LIN {X 0,Y 358.362,Z 472.331,A -85,B 0,C 180,E1 -13392.156,E2 -13392.156} C_VEL
LIN {X 0,Y 357.855,Z 480.13,A -85,B 0,C 180,E1 -13393.015,E2 -13393.015} C_VEL
LIN {X 0,Y 356.562,Z 489.991,A -85,B 0,C 180,E1 -13394.276,E2 -13394.276} C_VEL
LIN {X 0,Y 355.505,Z 499.646,A -85,B 0,C 180,E1 -13395.781,E2 -13395.781} C_VEL
LIN {X 0,Y 355.018,Z 505.416,A -85,B 0,C 180,E1 -13396.841,E2 -13396.841} C_VEL
LIN {X 0,Y 354.311,Z 513.334,A -85,B 0,C 180,E1 -13398.559,E2 -13398.559} C_VEL
LIN {X 0,Y 353.919,Z 519.825,A -85,B 0,C 180,E1 -13400.283,E2 -13400.283} C_VEL
LIN {X 0,Y 353.818,Z 525.056,A -85,B 0,C 180,E1 -13402.008,E2 -13402.008} C_VEL
LIN {X 0,Y 353.937,Z 528.669,A -85,B 0,C 180,E1 -13403.503,E2 -13403.503} C_VEL
LIN {X 0,Y 354.156,Z 532.195,A -85,B 0,C 180,E1 -13405.447,E2 -13405.447} C_VEL
LIN {X 0,Y 354.254,Z 533.682,A -85,B 0,C 180,E1 -13406.588,E2 -13406.588} C_VEL
LIN {X 0,Y 354.319,Z 534.699,A -85,B 0,C 180,E1 -13407.727,E2 -13407.727} C_VEL
LIN {X 0,Y 354.65,Z 535.319,A -85,B 0,C 180,E1 -13408.865,E2 -13408.865} C_VEL
LIN {X 0,Y 354.78,Z 535.5,A -85,B 0,C 180,E1 -13410,E2 -13410} C_VEL
LIN {X 0,Y 354.651,Z 535.226,A -85,B 0,C 180,E1 -13411.135,E2 -13411.135} C_VEL
LIN {X 0,Y 354.359,Z 534.457,A -85,B 0,C 180,E1 -13412.273,E2 -13412.273} C_VEL
LIN {X 0,Y 354.31,Z 533.29,A -85,B 0,C 180,E1 -13413.411,E2 -13413.411} C_VEL
LIN {X 0,Y 354.165,Z 530.683,A -85,B 0,C 180,E1 -13415.123,E2 -13415.123} C_VEL
LIN {X 0,Y 353.996,Z 526.732,A -85,B 0,C 180,E1 -13416.941,E2 -13416.941} C_VEL
LIN {X 0,Y 353.922,Z 522.099,A -85,B 0,C 180,E1 -13418.565,E2 -13418.565} C_VEL
LIN {X 0,Y 354.064,Z 515.923,A -85,B 0,C 180,E1 -13420.291,E2 -13420.291} C_VEL
LIN {X 0,Y 354.504,Z 508.22,A -85,B 0,C 180,E1 -13422.014,E2 -13422.014} C_VEL
LIN {X 0,Y 355.133,Z 500.362,A -85,B 0,C 180,E1 -13423.446,E2 -13423.446} C_VEL
LIN {X 0,Y 355.912,Z 490.818,A -85,B 0,C 180,E1 -13424.874,E2 -13424.874} C_VEL
LIN {X 0,Y 356.895,Z 480.343,A -85,B 0,C 180,E1 -13426.149,E2 -13426.149} C_VEL
LIN {X 0,Y 357.392,Z 473.331,A -85,B 0,C 180,E1 -13426.861,E2 -13426.861} C_VEL
LIN {X 0,Y 356.949,Z 460.178,A -85,B 0,C 180,E1 -13427.991,E2 -13427.991} C_VEL
LIN {X 0,Y 356.126,Z 447.743,A -85,B 0,C 180,E1 -13428.815,E2 -13428.815} C_VEL
LIN {X 0,Y 354.927,Z 433.651,A -85,B 0,C 180,E1 -13429.509,E2 -13429.509} C_VEL
LIN {X 0,Y 354.262,Z 426.541,A -85,B 0,C 180,E1 -13429.822,E2 -13429.822} C_VEL
LIN {X 0,Y 354.936,Z 413.74,A -85,B 0,C 180,E1 -13433.879,E2 -13433.879} C_VEL
LIN {X 0,Y 355.803,Z 401.985,A -85,B 0,C 180,E1 -13437.703,E2 -13437.703} C_VEL
LIN {X 0,Y 356.859,Z 390.592,A -85,B 0,C 180,E1 -13441.458,E2 -13441.458} C_VEL
LIN {X 0,Y 358.142,Z 378.993,A -85,B 0,C 180,E1 -13445.372,E2 -13445.372} C_VEL
LIN {X 0,Y 358.881,Z 373.147,A -85,B 0,C 180,E1 -13447.377,E2 -13447.377} C_VEL
LIN {X 0,Y 357.713,Z 366.126,A -85,B 0,C 180,E1 -13449.983,E2 -13449.983} C_VEL
LIN {X 0,Y 355.825,Z 356.518,A -85,B 0,C 180,E1 -13453.731,E2 -13453.731} C_VEL
LIN {X 0,Y 354.834,Z 351.339,A -85,B 0,C 180,E1 -13455.939,E2 -13455.939} C_VEL
LIN {X 0,Y 354.76,Z 351.295,A -85,B 0,C 180,E1 -13459.175,E2 -13459.175} C_VEL
LIN {X 0,Y 354.795,Z 351.287,A -85,B 0,C 180,E1 -13462.403,E2 -13462.403} C_VEL
LIN {X 0,Y 354.806,Z 351.288,A -85,B 0,C 180,E1 -13464.94,E2 -13464.94} C_VEL
LIN {X 0,Y 354.787,Z 351.288,A -85,B 0,C 180,E1 -13468.405,E2 -13468.405} C_VEL
LIN {X 0,Y 354.843,Z 351.283,A -85,B 0,C 180,E1 -13471.618,E2 -13471.618} C_VEL
LIN {X 0,Y 354.891,Z 351.275,A -85,B 0,C 180,E1 -13474.172,E2 -13474.172} C_VEL
LIN {X 0,Y 354.808,Z 351.285,A -85,B 0,C 180,E1 -13477.892,E2 -13477.892} C_VEL
LIN {X 0,Y 354.882,Z 351.276,A -85,B 0,C 180,E1 -13481.908,E2 -13481.908} C_VEL
LIN {X 0,Y 354.934,Z 351.269,A -85,B 0,C 180,E1 -13485.981,E2 -13485.981} C_VEL
LIN {X 0,Y 354.947,Z 351.268,A -85,B 0,C 180,E1 -13489.735,E2 -13489.735} C_VEL
LIN {X 0,Y 355.102,Z 351.252,A -85,B 0,C 180,E1 -13493.18,E2 -13493.18} C_VEL
LIN {X 0,Y 355.234,Z 351.232,A -85,B 0,C 180,E1 -13497.732,E2 -13497.732} C_VEL
LIN {X 0,Y 355.388,Z 351.213,A -85,B 0,C 180,E1 -13500,E2 -13500} C_VEL
LIN {X 0,Y 355.233,Z 351.234,A -85,B 0,C 180,E1 -13502.268,E2 -13502.268} C_VEL
LIN {X 0,Y 355.118,Z 351.252,A -85,B 0,C 180,E1 -13506.82,E2 -13506.82} C_VEL
LIN {X 0,Y 354.969,Z 351.267,A -85,B 0,C 180,E1 -13510.264,E2 -13510.264} C_VEL
LIN {X 0,Y 354.934,Z 351.27,A -85,B 0,C 180,E1 -13514.019,E2 -13514.019} C_VEL
LIN {X 0,Y 354.915,Z 351.274,A -85,B 0,C 180,E1 -13518.109,E2 -13518.109} C_VEL
LIN {X 0,Y 354.828,Z 351.285,A -85,B 0,C 180,E1 -13522.107,E2 -13522.107} C_VEL
LIN {X 0,Y 354.892,Z 351.276,A -85,B 0,C 180,E1 -13525.828,E2 -13525.828} C_VEL
LIN {X 0,Y 354.848,Z 351.281,A -85,B 0,C 180,E1 -13529.679,E2 -13529.679} C_VEL
LIN {X 0,Y 354.8,Z 351.287,A -85,B 0,C 180,E1 -13533.703,E2 -13533.703} C_VEL
LIN {X 0,Y 354.794,Z 351.291,A -85,B 0,C 180,E1 -13536.46,E2 -13536.46} C_VEL
LIN {X 0,Y 354.819,Z 351.284,A -85,B 0,C 180,E1 -13539.424,E2 -13539.424} C_VEL
LIN {X 0,Y 354.8,Z 351.287,A -85,B 0,C 180,E1 -13542.871,E2 -13542.871} C_VEL
LIN {X 0,Y 354.772,Z 351.295,A -85,B 0,C 180,E1 -13546.106,E2 -13546.106} C_VEL
LIN {X 0,Y 354.788,Z 351.288,A -85,B 0,C 180,E1 -13549.18,E2 -13549.18} C_VEL
LIN {X 0,Y 354.806,Z 351.288,A -85,B 0,C 180,E1 -13552.403,E2 -13552.403} C_VEL
LIN {X 0,Y 354.811,Z 351.285,A -85,B 0,C 180,E1 -13554.942,E2 -13554.942} C_VEL
LIN {X 0,Y 354.814,Z 351.287,A -85,B 0,C 180,E1 -13558.4,E2 -13558.4} C_VEL
LIN {X 0,Y 354.853,Z 351.282,A -85,B 0,C 180,E1 -13561.62,E2 -13561.62} C_VEL
LIN {X 0,Y 354.899,Z 351.277,A -85,B 0,C 180,E1 -13564.173,E2 -13564.173} C_VEL
LIN {X 0,Y 354.835,Z 351.288,A -85,B 0,C 180,E1 -13567.895,E2 -13567.895} C_VEL
LIN {X 0,Y 354.924,Z 351.276,A -85,B 0,C 180,E1 -13571.892,E2 -13571.892} C_VEL
LIN {X 0,Y 354.944,Z 351.272,A -85,B 0,C 180,E1 -13575.981,E2 -13575.981} C_VEL
LIN {X 0,Y 354.98,Z 351.27,A -85,B 0,C 180,E1 -13579.736,E2 -13579.736} C_VEL
LIN {X 0,Y 355.116,Z 351.249,A -85,B 0,C 180,E1 -13582.037,E2 -13582.037} C_VEL
LIN {X 0,Y 355.096,Z 351.25,A -85,B 0,C 180,E1 -13584.321,E2 -13584.321} C_VEL
LIN {X 0,Y 355.248,Z 351.235,A -85,B 0,C 180,E1 -13587.732,E2 -13587.732} C_VEL
LIN {X 0,Y 355.4,Z 351.213,A -85,B 0,C 180,E1 -13590,E2 -13590} C_VEL
LIN {X 0,Y 355.249,Z 351.231,A -85,B 0,C 180,E1 -13592.268,E2 -13592.268} C_VEL
LIN {X 0,Y 355.127,Z 351.246,A -85,B 0,C 180,E1 -13596.819,E2 -13596.819} C_VEL
LIN {X 0,Y 354.98,Z 351.264,A -85,B 0,C 180,E1 -13600.264,E2 -13600.264} C_VEL
LIN {X 0,Y 354.944,Z 351.269,A -85,B 0,C 180,E1 -13604.019,E2 -13604.019} C_VEL
LIN {X 0,Y 354.923,Z 351.271,A -85,B 0,C 180,E1 -13608.108,E2 -13608.108} C_VEL
LIN {X 0,Y 354.835,Z 351.282,A -85,B 0,C 180,E1 -13612.105,E2 -13612.105} C_VEL
LIN {X 0,Y 354.899,Z 351.275,A -85,B 0,C 180,E1 -13615.827,E2 -13615.827} C_VEL
LIN {X 0,Y 354.817,Z 351.285,A -85,B 0,C 180,E1 -13619.681,E2 -13619.681} C_VEL
LIN {X 0,Y 354.804,Z 351.286,A -85,B 0,C 180,E1 -13623.701,E2 -13623.701} C_VEL
LIN {X 0,Y 354.8,Z 351.287,A -85,B 0,C 180,E1 -13626.458,E2 -13626.458} C_VEL
LIN {X 0,Y 354.821,Z 351.287,A -85,B 0,C 180,E1 -13629.423,E2 -13629.423} C_VEL
LIN {X 0,Y 354.863,Z 351.283,A -85,B 0,C 180,E1 -13632.88,E2 -13632.88} C_VEL
LIN {X 0,Y 354.916,Z 351.438,A -85,B 0,C 180,E1 -13633.417,E2 -13633.417} C_VEL
LIN {X 0,Y 355.205,Z 352.666,A -85,B 0,C 180,E1 -13633.637,E2 -13633.637} C_VEL
LIN {X 0,Y 358.7,Z 364.873,A -85,B 0,C 180,E1 -13634.725,E2 -13634.725} C_VEL
LIN {X 0,Y 360.105,Z 371.17,A -85,B 0,C 180,E1 -13635.364,E2 -13635.364} C_VEL
LIN {X 0,Y 359.332,Z 381.796,A -85,B 0,C 180,E1 -13636.463,E2 -13636.463} C_VEL
LIN {X 0,Y 358.503,Z 392.374,A -85,B 0,C 180,E1 -13637.823,E2 -13637.823} C_VEL
LIN {X 0,Y 357.866,Z 399.364,A -85,B 0,C 180,E1 -13638.893,E2 -13638.893} C_VEL
LIN {X 0,Y 356.907,Z 403.436,A -85,B 0,C 180,E1 -13639.571,E2 -13639.571} C_VEL
LIN {X 0,Y 353.622,Z 409.736,A -85,B 0,C 180,E1 -13640.678,E2 -13640.678} C_VEL
LIN {X 0,Y 350.29,Z 415.539,A -85,B 0,C 180,E1 -13641.869,E2 -13641.869} C_VEL
LIN {X 0,Y 349.276,Z 418.689,A -85,B 0,C 180,E1 -13642.67,E2 -13642.67} C_VEL
LIN {X 0,Y 348.734,Z 423.802,A -85,B 0,C 180,E1 -13644.237,E2 -13644.237} C_VEL
LIN {X 0,Y 348.313,Z 429.257,A -85,B 0,C 180,E1 -13646.391,E2 -13646.391} C_VEL
LIN {X 0,Y 348.034,Z 432.759,A -85,B 0,C 180,E1 -13648.33,E2 -13648.33} C_VEL
LIN {X 0,Y 347.912,Z 435.084,A -85,B 0,C 180,E1 -13650.296,E2 -13650.296} C_VEL
LIN {X 0,Y 347.965,Z 436.386,A -85,B 0,C 180,E1 -13652.706,E2 -13652.706} C_VEL
LIN {X 0,Y 348.247,Z 436.007,A -85,B 0,C 180,E1 -13654.925,E2 -13654.925} C_VEL
LIN {X 0,Y 348.528,Z 435.142,A -85,B 0,C 180,E1 -13656.216,E2 -13656.216} C_VEL
LIN {X 0,Y 348.981,Z 433.251,A -85,B 0,C 180,E1 -13657.873,E2 -13657.873} C_VEL
LIN {X 0,Y 349.767,Z 429.478,A -85,B 0,C 180,E1 -13660.026,E2 -13660.026} C_VEL
LIN {X 0,Y 350.61,Z 424.843,A -85,B 0,C 180,E1 -13661.899,E2 -13661.899} C_VEL
LIN {X 0,Y 351.666,Z 418.867,A -85,B 0,C 180,E1 -13663.752,E2 -13663.752} C_VEL
LIN {X 0,Y 352.692,Z 412.681,A -85,B 0,C 180,E1 -13665.282,E2 -13665.282} C_VEL
LIN {X 0,Y 353.995,Z 404.139,A -85,B 0,C 180,E1 -13666.984,E2 -13666.984} C_VEL
LIN {X 0,Y 355.367,Z 393.993,A -85,B 0,C 180,E1 -13668.594,E2 -13668.594} C_VEL
LIN {X 0,Y 356.593,Z 383.387,A -85,B 0,C 180,E1 -13669.928,E2 -13669.928} C_VEL
LIN {X 0,Y 357.097,Z 377.92,A -85,B 0,C 180,E1 -13670.512,E2 -13670.512} C_VEL
LIN {X 0,Y 353.861,Z 367.207,A -85,B 0,C 180,E1 -13671.865,E2 -13671.865} C_VEL
LIN {X 0,Y 350.27,Z 357.755,A -85,B 0,C 180,E1 -13672.941,E2 -13672.941} C_VEL
LIN {X 0,Y 348.165,Z 352.79,A -85,B 0,C 180,E1 -13673.517,E2 -13673.517} C_VEL
LIN {X 0,Y 348.064,Z 352.162,A -85,B 0,C 180,E1 -13673.769,E2 -13673.769} C_VEL
LIN {X 0,Y 348.196,Z 352.114,A -85,B 0,C 180,E1 -13677.686,E2 -13677.686} C_VEL
LIN {X 0,Y 348.337,Z 352.096,A -85,B 0,C 180,E1 -13680,E2 -13680} C_VEL
LIN {X 0,Y 348.196,Z 352.112,A -85,B 0,C 180,E1 -13682.314,E2 -13682.314} C_VEL
LIN {X 0,Y 348.068,Z 352.128,A -85,B 0,C 180,E1 -13686.958,E2 -13686.958} C_VEL
LIN {X 0,Y 347.887,Z 352.149,A -85,B 0,C 180,E1 -13690.476,E2 -13690.476} C_VEL
LIN {X 0,Y 347.891,Z 352.149,A -85,B 0,C 180,E1 -13694.15,E2 -13694.15} C_VEL
LIN {X 0,Y 347.821,Z 352.154,A -85,B 0,C 180,E1 -13698.26,E2 -13698.26} C_VEL
LIN {X 0,Y 347.76,Z 352.166,A -85,B 0,C 180,E1 -13701.627,E2 -13701.627} C_VEL
LIN {X 0,Y 347.805,Z 352.163,A -85,B 0,C 180,E1 -13705.109,E2 -13705.109} C_VEL
LIN {X 0,Y 347.802,Z 352.162,A -85,B 0,C 180,E1 -13707.695,E2 -13707.695} C_VEL
LIN {X 0,Y 347.743,Z 352.171,A -85,B 0,C 180,E1 -13710.349,E2 -13710.349} C_VEL
LIN {X 0,Y 347.743,Z 352.169,A -85,B 0,C 180,E1 -13714.045,E2 -13714.045} C_VEL
LIN {X 0,Y 347.751,Z 352.168,A -85,B 0,C 180,E1 -13717.322,E2 -13717.322} C_VEL
LIN {X 0,Y 347.734,Z 352.185,A -85,B 0,C 180,E1 -13721.601,E2 -13721.601} C_VEL
LIN {X 0,Y 348.038,Z 353.526,A -85,B 0,C 180,E1 -13722.569,E2 -13722.569} C_VEL
LIN {X 0,Y 349.523,Z 360.428,A -85,B 0,C 180,E1 -13726.375,E2 -13726.375} C_VEL
LIN {X 0,Y 351.027,Z 368.334,A -85,B 0,C 180,E1 -13730.159,E2 -13730.159} C_VEL
LIN {X 0,Y 351.776,Z 373.684,A -85,B 0,C 180,E1 -13732.46,E2 -13732.46} C_VEL
LIN {X 0,Y 350.204,Z 384.504,A -85,B 0,C 180,E1 -13736.505,E2 -13736.505} C_VEL
LIN {X 0,Y 349.147,Z 394.206,A -85,B 0,C 180,E1 -13739.946,E2 -13739.946} C_VEL
LIN {X 0,Y 348.219,Z 405.075,A -85,B 0,C 180,E1 -13743.64,E2 -13743.64} C_VEL
LIN {X 0,Y 347.447,Z 417.359,A -85,B 0,C 180,E1 -13747.625,E2 -13747.625} C_VEL
LIN {X 0,Y 347.592,Z 419.174,A -85,B 0,C 180,E1 -13747.812,E2 -13747.812} C_VEL
LIN {X 0,Y 350.112,Z 432.508,A -85,B 0,C 180,E1 -13748.583,E2 -13748.583} C_VEL
LIN {X 0,Y 351.458,Z 445.441,A -85,B 0,C 180,E1 -13749.441,E2 -13749.441} C_VEL
LIN {X 0,Y 351.882,Z 457.391,A -85,B 0,C 180,E1 -13750.379,E2 -13750.379} C_VEL
LIN {X 0,Y 351.551,Z 469.302,A -85,B 0,C 180,E1 -13751.497,E2 -13751.497} C_VEL
LIN {X 0,Y 351.215,Z 478.527,A -85,B 0,C 180,E1 -13752.533,E2 -13752.533} C_VEL
LIN {X 0,Y 349.667,Z 489.454,A -85,B 0,C 180,E1 -13753.957,E2 -13753.957} C_VEL
LIN {X 0,Y 348.568,Z 498.626,A -85,B 0,C 180,E1 -13755.421,E2 -13755.421} C_VEL
LIN {X 0,Y 348.085,Z 504.722,A -85,B 0,C 180,E1 -13756.574,E2 -13756.574} C_VEL
LIN {X 0,Y 347.306,Z 512.567,A -85,B 0,C 180,E1 -13758.325,E2 -13758.325} C_VEL
LIN {X 0,Y 346.847,Z 518.982,A -85,B 0,C 180,E1 -13760.083,E2 -13760.083} C_VEL
LIN {X 0,Y 346.74,Z 524.165,A -85,B 0,C 180,E1 -13761.843,E2 -13761.843} C_VEL
LIN {X 0,Y 346.825,Z 527.351,A -85,B 0,C 180,E1 -13763.183,E2 -13763.183} C_VEL
LIN {X 0,Y 347.091,Z 531.243,A -85,B 0,C 180,E1 -13765.354,E2 -13765.354} C_VEL
LIN {X 0,Y 347.203,Z 532.71,A -85,B 0,C 180,E1 -13766.519,E2 -13766.519} C_VEL
LIN {X 0,Y 347.617,Z 534.301,A -85,B 0,C 180,E1 -13768.842,E2 -13768.842} C_VEL
LIN {X 0,Y 347.772,Z 534.47,A -85,B 0,C 180,E1 -13770,E2 -13770} C_VEL
LIN {X 0,Y 347.621,Z 534.165,A -85,B 0,C 180,E1 -13771.158,E2 -13771.158} C_VEL
LIN {X 0,Y 347.27,Z 532.179,A -85,B 0,C 180,E1 -13773.481,E2 -13773.481} C_VEL
LIN {X 0,Y 347.108,Z 529.527,A -85,B 0,C 180,E1 -13775.228,E2 -13775.228} C_VEL
LIN {X 0,Y 346.945,Z 525.775,A -85,B 0,C 180,E1 -13776.981,E2 -13776.981} C_VEL
LIN {X 0,Y 346.874,Z 520.839,A -85,B 0,C 180,E1 -13778.74,E2 -13778.74} C_VEL
LIN {X 0,Y 347.015,Z 514.6,A -85,B 0,C 180,E1 -13780.502,E2 -13780.502} C_VEL
LIN {X 0,Y 347.491,Z 506.787,A -85,B 0,C 180,E1 -13782.261,E2 -13782.261} C_VEL
LIN {X 0,Y 348.101,Z 498.832,A -85,B 0,C 180,E1 -13783.723,E2 -13783.723} C_VEL
LIN {X 0,Y 348.98,Z 489.198,A -85,B 0,C 180,E1 -13785.177,E2 -13785.177} C_VEL
LIN {X 0,Y 350.007,Z 478.575,A -85,B 0,C 180,E1 -13786.476,E2 -13786.476} C_VEL
LIN {X 0,Y 350.321,Z 472.921,A -85,B 0,C 180,E1 -13787.061,E2 -13787.061} C_VEL
LIN {X 0,Y 349.964,Z 460.881,A -85,B 0,C 180,E1 -13788.135,E2 -13788.135} C_VEL
LIN {X 0,Y 349.245,Z 449.494,A -85,B 0,C 180,E1 -13788.95,E2 -13788.95} C_VEL
LIN {X 0,Y 348.207,Z 435.937,A -85,B 0,C 180,E1 -13789.682,E2 -13789.682} C_VEL
LIN {X 0,Y 347.223,Z 425.817,A -85,B 0,C 180,E1 -13790.126,E2 -13790.126} C_VEL
LIN {X 0,Y 347.596,Z 418.073,A -85,B 0,C 180,E1 -13792.591,E2 -13792.591} C_VEL
LIN {X 0,Y 348.391,Z 406.693,A -85,B 0,C 180,E1 -13796.346,E2 -13796.346} C_VEL
LIN {X 0,Y 349.398,Z 395.257,A -85,B 0,C 180,E1 -13800.189,E2 -13800.189} C_VEL
LIN {X 0,Y 350.427,Z 385.651,A -85,B 0,C 180,E1 -13803.471,E2 -13803.471} C_VEL
LIN {X 0,Y 351.762,Z 375.625,A -85,B 0,C 180,E1 -13806.948,E2 -13806.948} C_VEL
LIN {X 0,Y 351.777,Z 372.982,A -85,B 0,C 180,E1 -13807.904,E2 -13807.904} C_VEL
LIN {X 0,Y 350.001,Z 363.655,A -85,B 0,C 180,E1 -13811.5,E2 -13811.5} C_VEL
LIN {X 0,Y 348.319,Z 354.848,A -85,B 0,C 180,E1 -13815.074,E2 -13815.074} C_VEL
LIN {X 0,Y 347.758,Z 352.252,A -85,B 0,C 180,E1 -13816.197,E2 -13816.197} C_VEL
LIN {X 0,Y 347.692,Z 352.174,A -85,B 0,C 180,E1 -13819.697,E2 -13819.697} C_VEL
LIN {X 0,Y 347.751,Z 352.165,A -85,B 0,C 180,E1 -13822.678,E2 -13822.678} C_VEL
LIN {X 0,Y 347.743,Z 352.166,A -85,B 0,C 180,E1 -13825.955,E2 -13825.955} C_VEL
LIN {X 0,Y 347.758,Z 352.165,A -85,B 0,C 180,E1 -13829.653,E2 -13829.653} C_VEL
LIN {X 0,Y 347.844,Z 352.155,A -85,B 0,C 180,E1 -13832.744,E2 -13832.744} C_VEL
LIN {X 0,Y 347.778,Z 352.161,A -85,B 0,C 180,E1 -13836.161,E2 -13836.161} C_VEL
LIN {X 0,Y 347.792,Z 352.159,A -85,B 0,C 180,E1 -13839.908,E2 -13839.908} C_VEL
LIN {X 0,Y 347.824,Z 352.157,A -85,B 0,C 180,E1 -13843.568,E2 -13843.568} C_VEL
LIN {X 0,Y 347.881,Z 352.152,A -85,B 0,C 180,E1 -13847.16,E2 -13847.16} C_VEL
LIN {X 0,Y 347.927,Z 352.146,A -85,B 0,C 180,E1 -13850.7,E2 -13850.7} C_VEL
LIN {X 0,Y 348.068,Z 352.129,A -85,B 0,C 180,E1 -13853.042,E2 -13853.042} C_VEL
LIN {X 0,Y 348.196,Z 352.109,A -85,B 0,C 180,E1 -13857.686,E2 -13857.686} C_VEL
LIN {X 0,Y 348.337,Z 352.091,A -85,B 0,C 180,E1 -13860,E2 -13860} C_VEL
LIN {X 0,Y 348.196,Z 352.111,A -85,B 0,C 180,E1 -13862.314,E2 -13862.314} C_VEL
LIN {X 0,Y 348.084,Z 352.126,A -85,B 0,C 180,E1 -13866.958,E2 -13866.958} C_VEL
LIN {X 0,Y 347.92,Z 352.147,A -85,B 0,C 180,E1 -13870.475,E2 -13870.475} C_VEL
LIN {X 0,Y 347.891,Z 352.149,A -85,B 0,C 180,E1 -13874.15,E2 -13874.15} C_VEL
LIN {X 0,Y 347.884,Z 352.151,A -85,B 0,C 180,E1 -13878.291,E2 -13878.291} C_VEL
LIN {X 0,Y 347.782,Z 352.16,A -85,B 0,C 180,E1 -13881.636,E2 -13881.636} C_VEL
LIN {X 0,Y 347.805,Z 352.158,A -85,B 0,C 180,E1 -13885.109,E2 -13885.109} C_VEL
LIN {X 0,Y 347.806,Z 352.158,A -85,B 0,C 180,E1 -13887.694,E2 -13887.694} C_VEL
LIN {X 0,Y 347.758,Z 352.169,A -85,B 0,C 180,E1 -13890.347,E2 -13890.347} C_VEL
LIN {X 0,Y 347.739,Z 352.17,A -85,B 0,C 180,E1 -13894.465,E2 -13894.465} C_VEL
LIN {X 0,Y 347.77,Z 352.165,A -85,B 0,C 180,E1 -13897.99,E2 -13897.99} C_VEL
LIN {X 0,Y 347.762,Z 352.165,A -85,B 0,C 180,E1 -13901.829,E2 -13901.829} C_VEL
LIN {X 0,Y 347.73,Z 352.167,A -85,B 0,C 180,E1 -13905.023,E2 -13905.023} C_VEL
LIN {X 0,Y 347.75,Z 352.168,A -85,B 0,C 180,E1 -13908.397,E2 -13908.397} C_VEL
LIN {X 0,Y 347.772,Z 352.167,A -85,B 0,C 180,E1 -13912.012,E2 -13912.012} C_VEL
LIN {X 0,Y 347.743,Z 352.167,A -85,B 0,C 180,E1 -13915.537,E2 -13915.537} C_VEL
LIN {X 0,Y 347.763,Z 352.166,A -85,B 0,C 180,E1 -13918.303,E2 -13918.303} C_VEL
LIN {X 0,Y 347.805,Z 352.157,A -85,B 0,C 180,E1 -13920.991,E2 -13920.991} C_VEL
LIN {X 0,Y 347.832,Z 352.157,A -85,B 0,C 180,E1 -13923.609,E2 -13923.609} C_VEL
LIN {X 0,Y 347.789,Z 352.163,A -85,B 0,C 180,E1 -13926.163,E2 -13926.163} C_VEL
LIN {X 0,Y 347.818,Z 352.161,A -85,B 0,C 180,E1 -13929.91,E2 -13929.91} C_VEL
LIN {X 0,Y 347.868,Z 352.151,A -85,B 0,C 180,E1 -13932.36,E2 -13932.36} C_VEL
LIN {X 0,Y 347.899,Z 352.15,A -85,B 0,C 180,E1 -13935.971,E2 -13935.971} C_VEL
LIN {X 0,Y 347.931,Z 352.146,A -85,B 0,C 180,E1 -13939.526,E2 -13939.526} C_VEL
LIN {X 0,Y 348.077,Z 352.128,A -85,B 0,C 180,E1 -13941.875,E2 -13941.875} C_VEL
LIN {X 0,Y 348.071,Z 352.125,A -85,B 0,C 180,E1 -13944.206,E2 -13944.206} C_VEL
LIN {X 0,Y 348.211,Z 352.112,A -85,B 0,C 180,E1 -13947.687,E2 -13947.687} C_VEL
LIN {X 0,Y 348.37,Z 352.089,A -85,B 0,C 180,E1 -13950,E2 -13950} C_VEL
LIN {X 0,Y 348.211,Z 352.107,A -85,B 0,C 180,E1 -13952.313,E2 -13952.313} C_VEL
LIN {X 0,Y 348.093,Z 352.123,A -85,B 0,C 180,E1 -13956.958,E2 -13956.958} C_VEL
LIN {X 0,Y 347.931,Z 352.142,A -85,B 0,C 180,E1 -13960.474,E2 -13960.474} C_VEL
LIN {X 0,Y 347.9,Z 352.146,A -85,B 0,C 180,E1 -13964.149,E2 -13964.149} C_VEL
LIN {X 0,Y 347.891,Z 352.147,A -85,B 0,C 180,E1 -13968.29,E2 -13968.29} C_VEL
LIN {X 0,Y 347.789,Z 352.162,A -85,B 0,C 180,E1 -13971.635,E2 -13971.635} C_VEL
LIN {X 0,Y 347.813,Z 352.162,A -85,B 0,C 180,E1 -13975.108,E2 -13975.108} C_VEL
LIN {X 0,Y 347.807,Z 352.159,A -85,B 0,C 180,E1 -13977.693,E2 -13977.693} C_VEL
LIN {X 0,Y 347.748,Z 352.165,A -85,B 0,C 180,E1 -13980.347,E2 -13980.347} C_VEL
LIN {X 0,Y 347.746,Z 352.165,A -85,B 0,C 180,E1 -13984.043,E2 -13984.043} C_VEL
LIN {X 0,Y 347.765,Z 352.166,A -85,B 0,C 180,E1 -13987.319,E2 -13987.319} C_VEL
LIN {X 0,Y 347.791,Z 352.164,A -85,B 0,C 180,E1 -13990.288,E2 -13990.288} C_VEL
LIN {X 0,Y 347.848,Z 352.299,A -85,B 0,C 180,E1 -13993.111,E2 -13993.111} C_VEL
LIN {X 0,Y 348.15,Z 353.58,A -85,B 0,C 180,E1 -13993.34,E2 -13993.34} C_VEL
LIN {X 0,Y 351.892,Z 366.568,A -85,B 0,C 180,E1 -13994.531,E2 -13994.531} C_VEL
LIN {X 0,Y 353.126,Z 371.448,A -85,B 0,C 180,E1 -13995.043,E2 -13995.043} C_VEL
LIN {X 0,Y 352.491,Z 382.216,A -85,B 0,C 180,E1 -13996.173,E2 -13996.173} C_VEL
LIN {X 0,Y 351.656,Z 392.654,A -85,B 0,C 180,E1 -13997.519,E2 -13997.519} C_VEL
LIN {X 0,Y 350.66,Z 403.079,A -85,B 0,C 180,E1 -13999.195,E2 -13999.195} C_VEL
LIN {X 0,Y 349.942,Z 410.961,A -85,B 0,C 180,E1 -14000.756,E2 -14000.756} C_VEL
LIN {X 0,Y 349.276,Z 418.689,A -85,B 0,C 180,E1 -14002.67,E2 -14002.67} C_VEL
LIN {X 0,Y 348.284,Z 421.652,A -85,B 0,C 180,E1 -14003.496,E2 -14003.496} C_VEL
LIN {X 0,Y 345.055,Z 426.138,A -85,B 0,C 180,E1 -14004.857,E2 -14004.857} C_VEL
LIN {X 0,Y 341.939,Z 429.996,A -85,B 0,C 180,E1 -14006.291,E2 -14006.291} C_VEL
LIN {X 0,Y 341.141,Z 431.89,A -85,B 0,C 180,E1 -14007.22,E2 -14007.22} C_VEL
LIN {X 0,Y 340.934,Z 434.654,A -85,B 0,C 180,E1 -14008.979,E2 -14008.979} C_VEL
LIN {X 0,Y 340.892,Z 436.108,A -85,B 0,C 180,E1 -14010.344,E2 -14010.344} C_VEL
LIN {X 0,Y 340.932,Z 437.318,A -85,B 0,C 180,E1 -14012.422,E2 -14012.422} C_VEL
LIN {X 0,Y 341.25,Z 437.113,A -85,B 0,C 180,E1 -14014.979,E2 -14014.979} C_VEL
LIN {X 0,Y 341.72,Z 435.618,A -85,B 0,C 180,E1 -14016.998,E2 -14016.998} C_VEL
LIN {X 0,Y 342.378,Z 433.031,A -85,B 0,C 180,E1 -14018.947,E2 -14018.947} C_VEL
LIN {X 0,Y 343.134,Z 429.312,A -85,B 0,C 180,E1 -14020.87,E2 -14020.87} C_VEL
LIN {X 0,Y 344.15,Z 424.285,A -85,B 0,C 180,E1 -14022.776,E2 -14022.776} C_VEL
LIN {X 0,Y 345.316,Z 417.835,A -85,B 0,C 180,E1 -14024.658,E2 -14024.658} C_VEL
LIN {X 0,Y 346.607,Z 410.454,A -85,B 0,C 180,E1 -14026.366,E2 -14026.366} C_VEL
LIN {X 0,Y 347.695,Z 403.174,A -85,B 0,C 180,E1 -14027.746,E2 -14027.746} C_VEL
LIN {X 0,Y 349.151,Z 393.29,A -85,B 0,C 180,E1 -14029.269,E2 -14029.269} C_VEL
LIN {X 0,Y 350.355,Z 383.05,A -85,B 0,C 180,E1 -14030.547,E2 -14030.547} C_VEL
LIN {X 0,Y 350.561,Z 379.755,A -85,B 0,C 180,E1 -14030.916,E2 -14030.916} C_VEL
LIN {X 0,Y 347.544,Z 369.665,A -85,B 0,C 180,E1 -14032.243,E2 -14032.243} C_VEL
LIN {X 0,Y 343.446,Z 358.895,A -85,B 0,C 180,E1 -14033.538,E2 -14033.538} C_VEL
LIN {X 0,Y 341.156,Z 353.736,A -85,B 0,C 180,E1 -14034.162,E2 -14034.162} C_VEL
LIN {X 0,Y 340.96,Z 353.046,A -85,B 0,C 180,E1 -14034.455,E2 -14034.455} C_VEL
LIN {X 0,Y 341.158,Z 352.99,A -85,B 0,C 180,E1 -14037.639,E2 -14037.639} C_VEL
LIN {X 0,Y 341.287,Z 352.975,A -85,B 0,C 180,E1 -14040,E2 -14040} C_VEL
LIN {X 0,Y 341.158,Z 352.989,A -85,B 0,C 180,E1 -14042.361,E2 -14042.361} C_VEL
LIN {X 0,Y 341.036,Z 353.005,A -85,B 0,C 180,E1 -14047.103,E2 -14047.103} C_VEL
LIN {X 0,Y 340.839,Z 353.028,A -85,B 0,C 180,E1 -14050.695,E2 -14050.695} C_VEL
LIN {X 0,Y 340.856,Z 353.026,A -85,B 0,C 180,E1 -14054.325,E2 -14054.325} C_VEL
LIN {X 0,Y 340.779,Z 353.032,A -85,B 0,C 180,E1 -14058.441,E2 -14058.441} C_VEL
LIN {X 0,Y 340.711,Z 353.045,A -85,B 0,C 180,E1 -14061.842,E2 -14061.842} C_VEL
LIN {X 0,Y 340.765,Z 353.036,A -85,B 0,C 180,E1 -14065.665,E2 -14065.665} C_VEL
LIN {X 0,Y 340.722,Z 353.042,A -85,B 0,C 180,E1 -14068.321,E2 -14068.321} C_VEL
LIN {X 0,Y 340.691,Z 353.045,A -85,B 0,C 180,E1 -14071.045,E2 -14071.045} C_VEL
LIN {X 0,Y 340.712,Z 353.043,A -85,B 0,C 180,E1 -14075.28,E2 -14075.28} C_VEL
LIN {X 0,Y 340.688,Z 353.048,A -85,B 0,C 180,E1 -14078.383,E2 -14078.383} C_VEL
LIN {X 0,Y 340.688,Z 353.171,A -85,B 0,C 180,E1 -14081.015,E2 -14081.015} C_VEL
LIN {X 0,Y 341.886,Z 358.639,A -85,B 0,C 180,E1 -14084.341,E2 -14084.341} C_VEL
LIN {X 0,Y 343.106,Z 364.605,A -85,B 0,C 180,E1 -14087.511,E2 -14087.511} C_VEL
LIN {X 0,Y 344.414,Z 371.625,A -85,B 0,C 180,E1 -14090.843,E2 -14090.843} C_VEL
LIN {X 0,Y 344.845,Z 374.984,A -85,B 0,C 180,E1 -14092.31,E2 -14092.31} C_VEL
LIN {X 0,Y 343.225,Z 385.747,A -85,B 0,C 180,E1 -14096.437,E2 -14096.437} C_VEL
LIN {X 0,Y 341.96,Z 396.829,A -85,B 0,C 180,E1 -14100.446,E2 -14100.446} C_VEL
LIN {X 0,Y 340.994,Z 408.119,A -85,B 0,C 180,E1 -14104.354,E2 -14104.354} C_VEL
LIN {X 0,Y 340.457,Z 416.172,A -85,B 0,C 180,E1 -14107.005,E2 -14107.005} C_VEL
LIN {X 0,Y 340.648,Z 418.024,A -85,B 0,C 180,E1 -14107.171,E2 -14107.171} C_VEL
LIN {X 0,Y 343.135,Z 430.572,A -85,B 0,C 180,E1 -14107.933,E2 -14107.933} C_VEL
LIN {X 0,Y 344.667,Z 443.838,A -85,B 0,C 180,E1 -14108.86,E2 -14108.86} C_VEL
LIN {X 0,Y 345.119,Z 456.528,A -85,B 0,C 180,E1 -14109.884,E2 -14109.884} C_VEL
LIN {X 0,Y 344.816,Z 467.8,A -85,B 0,C 180,E1 -14110.968,E2 -14110.968} C_VEL
LIN {X 0,Y 344.26,Z 479.412,A -85,B 0,C 180,E1 -14112.322,E2 -14112.322} C_VEL
LIN {X 0,Y 342.839,Z 488.987,A -85,B 0,C 180,E1 -14113.629,E2 -14113.629} C_VEL
LIN {X 0,Y 341.569,Z 498.748,A -85,B 0,C 180,E1 -14115.253,E2 -14115.253} C_VEL
LIN {X 0,Y 340.929,Z 505.454,A -85,B 0,C 180,E1 -14116.591,E2 -14116.591} C_VEL
LIN {X 0,Y 340.177,Z 512.982,A -85,B 0,C 180,E1 -14118.38,E2 -14118.38} C_VEL
LIN {X 0,Y 339.713,Z 519.993,A -85,B 0,C 180,E1 -14120.474,E2 -14120.474} C_VEL
LIN {X 0,Y 339.675,Z 524.738,A -85,B 0,C 180,E1 -14122.271,E2 -14122.271} C_VEL
LIN {X 0,Y 339.829,Z 528.4,A -85,B 0,C 180,E1 -14124.065,E2 -14124.065} C_VEL
LIN {X 0,Y 340.027,Z 530.291,A -85,B 0,C 180,E1 -14125.258,E2 -14125.258} C_VEL
LIN {X 0,Y 340.153,Z 531.729,A -85,B 0,C 180,E1 -14126.446,E2 -14126.446} C_VEL
LIN {X 0,Y 340.583,Z 533.288,A -85,B 0,C 180,E1 -14128.818,E2 -14128.818} C_VEL
LIN {X 0,Y 340.762,Z 533.443,A -85,B 0,C 180,E1 -14130,E2 -14130} C_VEL
LIN {X 0,Y 340.59,Z 533.093,A -85,B 0,C 180,E1 -14131.182,E2 -14131.182} C_VEL
LIN {X 0,Y 340.229,Z 531.066,A -85,B 0,C 180,E1 -14133.553,E2 -14133.553} C_VEL
LIN {X 0,Y 340.052,Z 528.364,A -85,B 0,C 180,E1 -14135.336,E2 -14135.336} C_VEL
LIN {X 0,Y 339.877,Z 524.558,A -85,B 0,C 180,E1 -14137.127,E2 -14137.127} C_VEL
LIN {X 0,Y 339.806,Z 519.565,A -85,B 0,C 180,E1 -14138.923,E2 -14138.923} C_VEL
LIN {X 0,Y 339.996,Z 513.256,A -85,B 0,C 180,E1 -14140.721,E2 -14140.721} C_VEL
LIN {X 0,Y 340.489,Z 505.34,A -85,B 0,C 180,E1 -14142.517,E2 -14142.517} C_VEL
LIN {X 0,Y 341.099,Z 497.292,A -85,B 0,C 180,E1 -14144.01,E2 -14144.01} C_VEL
LIN {X 0,Y 342.102,Z 487.58,A -85,B 0,C 180,E1 -14145.489,E2 -14145.489} C_VEL
LIN {X 0,Y 343.213,Z 476.771,A -85,B 0,C 180,E1 -14146.812,E2 -14146.812} C_VEL
LIN {X 0,Y 343.116,Z 466.062,A -85,B 0,C 180,E1 -14147.893,E2 -14147.893} C_VEL
LIN {X 0,Y 342.501,Z 452.954,A -85,B 0,C 180,E1 -14148.959,E2 -14148.959} C_VEL
LIN {X 0,Y 341.51,Z 439.372,A -85,B 0,C 180,E1 -14149.791,E2 -14149.791} C_VEL
LIN {X 0,Y 340.184,Z 425.2,A -85,B 0,C 180,E1 -14150.442,E2 -14150.442} C_VEL
LIN {X 0,Y 340.176,Z 424.448,A -85,B 0,C 180,E1 -14150.561,E2 -14150.561} C_VEL
LIN {X 0,Y 340.849,Z 413.1,A -85,B 0,C 180,E1 -14154.354,E2 -14154.354} C_VEL
LIN {X 0,Y 341.777,Z 401.75,A -85,B 0,C 180,E1 -14158.225,E2 -14158.225} C_VEL
LIN {X 0,Y 342.945,Z 390.289,A -85,B 0,C 180,E1 -14162.195,E2 -14162.195} C_VEL
LIN {X 0,Y 344.636,Z 377.243,A -85,B 0,C 180,E1 -14166.815,E2 -14166.815} C_VEL
LIN {X 0,Y 344.851,Z 374.832,A -85,B 0,C 180,E1 -14167.689,E2 -14167.689} C_VEL
LIN {X 0,Y 343.352,Z 366.552,A -85,B 0,C 180,E1 -14170.918,E2 -14170.918} C_VEL
LIN {X 0,Y 341.719,Z 358.123,A -85,B 0,C 180,E1 -14174.367,E2 -14174.367} C_VEL
LIN {X 0,Y 340.724,Z 353.12,A -85,B 0,C 180,E1 -14176.557,E2 -14176.557} C_VEL
LIN {X 0,Y 340.65,Z 353.049,A -85,B 0,C 180,E1 -14180.24,E2 -14180.24} C_VEL
LIN {X 0,Y 340.703,Z 353.046,A -85,B 0,C 180,E1 -14183.559,E2 -14183.559} C_VEL
LIN {X 0,Y 340.687,Z 353.044,A -85,B 0,C 180,E1 -14186.153,E2 -14186.153} C_VEL
LIN {X 0,Y 340.768,Z 353.034,A -85,B 0,C 180,E1 -14190.332,E2 -14190.332} C_VEL
LIN {X 0,Y 340.797,Z 353.035,A -85,B 0,C 180,E1 -14193.019,E2 -14193.019} C_VEL
LIN {X 0,Y 340.747,Z 353.038,A -85,B 0,C 180,E1 -14195.638,E2 -14195.638} C_VEL
LIN {X 0,Y 340.722,Z 353.042,A -85,B 0,C 180,E1 -14199.472,E2 -14199.472} C_VEL
LIN {X 0,Y 340.784,Z 353.032,A -85,B 0,C 180,E1 -14201.98,E2 -14201.98} C_VEL
LIN {X 0,Y 340.862,Z 353.023,A -85,B 0,C 180,E1 -14205.705,E2 -14205.705} C_VEL
LIN {X 0,Y 340.839,Z 353.028,A -85,B 0,C 180,E1 -14209.305,E2 -14209.305} C_VEL
LIN {X 0,Y 341.036,Z 353.007,A -85,B 0,C 180,E1 -14212.897,E2 -14212.897} C_VEL
LIN {X 0,Y 341.158,Z 352.986,A -85,B 0,C 180,E1 -14217.639,E2 -14217.639} C_VEL
LIN {X 0,Y 341.287,Z 352.97,A -85,B 0,C 180,E1 -14220,E2 -14220} C_VEL
LIN {X 0,Y 341.157,Z 352.988,A -85,B 0,C 180,E1 -14222.361,E2 -14222.361} C_VEL
LIN {X 0,Y 341.052,Z 353.001,A -85,B 0,C 180,E1 -14227.102,E2 -14227.102} C_VEL
LIN {X 0,Y 340.862,Z 353.028,A -85,B 0,C 180,E1 -14230.694,E2 -14230.694} C_VEL
LIN {X 0,Y 340.856,Z 353.026,A -85,B 0,C 180,E1 -14234.325,E2 -14234.325} C_VEL
LIN {X 0,Y 340.831,Z 353.032,A -85,B 0,C 180,E1 -14238.467,E2 -14238.467} C_VEL
LIN {X 0,Y 340.747,Z 353.038,A -85,B 0,C 180,E1 -14241.857,E2 -14241.857} C_VEL
LIN {X 0,Y 340.766,Z 353.035,A -85,B 0,C 180,E1 -14245.665,E2 -14245.665} C_VEL
LIN {X 0,Y 340.736,Z 353.043,A -85,B 0,C 180,E1 -14248.32,E2 -14248.32} C_VEL
LIN {X 0,Y 340.698,Z 353.043,A -85,B 0,C 180,E1 -14251.045,E2 -14251.045} C_VEL
LIN {X 0,Y 340.713,Z 353.041,A -85,B 0,C 180,E1 -14255.28,E2 -14255.28} C_VEL
LIN {X 0,Y 340.708,Z 353.046,A -85,B 0,C 180,E1 -14258.387,E2 -14258.387} C_VEL
LIN {X 0,Y 340.725,Z 353.044,A -85,B 0,C 180,E1 -14262.052,E2 -14262.052} C_VEL
LIN {X 0,Y 340.658,Z 353.053,A -85,B 0,C 180,E1 -14266.226,E2 -14266.226} C_VEL
LIN {X 0,Y 340.688,Z 353.047,A -85,B 0,C 180,E1 -14269.753,E2 -14269.753} C_VEL
LIN {X 0,Y 340.703,Z 353.042,A -85,B 0,C 180,E1 -14273.259,E2 -14273.259} C_VEL
LIN {X 0,Y 340.694,Z 353.048,A -85,B 0,C 180,E1 -14276.154,E2 -14276.154} C_VEL
LIN {X 0,Y 340.775,Z 353.036,A -85,B 0,C 180,E1 -14280.333,E2 -14280.333} C_VEL
LIN {X 0,Y 340.805,Z 353.03,A -85,B 0,C 180,E1 -14283.021,E2 -14283.021} C_VEL
LIN {X 0,Y 340.729,Z 353.039,A -85,B 0,C 180,E1 -14286.928,E2 -14286.928} C_VEL
LIN {X 0,Y 340.796,Z 353.031,A -85,B 0,C 180,E1 -14290.734,E2 -14290.734} C_VEL
LIN {X 0,Y 340.789,Z 353.033,A -85,B 0,C 180,E1 -14293.219,E2 -14293.219} C_VEL
LIN {X 0,Y 340.846,Z 353.025,A -85,B 0,C 180,E1 -14296.891,E2 -14296.891} C_VEL
LIN {X 0,Y 340.93,Z 353.014,A -85,B 0,C 180,E1 -14300.508,E2 -14300.508} C_VEL
LIN {X 0,Y 341.078,Z 352.996,A -85,B 0,C 180,E1 -14302.898,E2 -14302.898} C_VEL
LIN {X 0,Y 341.172,Z 352.989,A -85,B 0,C 180,E1 -14307.639,E2 -14307.639} C_VEL
LIN {X 0,Y 341.319,Z 352.967,A -85,B 0,C 180,E1 -14310,E2 -14310} C_VEL
LIN {X 0,Y 341.173,Z 352.984,A -85,B 0,C 180,E1 -14312.361,E2 -14312.361} C_VEL
LIN {X 0,Y 341.061,Z 353,A -85,B 0,C 180,E1 -14317.102,E2 -14317.102} C_VEL
LIN {X 0,Y 340.873,Z 353.022,A -85,B 0,C 180,E1 -14320.693,E2 -14320.693} C_VEL
LIN {X 0,Y 340.864,Z 353.022,A -85,B 0,C 180,E1 -14324.324,E2 -14324.324} C_VEL
LIN {X 0,Y 340.838,Z 353.026,A -85,B 0,C 180,E1 -14328.466,E2 -14328.466} C_VEL
LIN {X 0,Y 340.754,Z 353.037,A -85,B 0,C 180,E1 -14331.856,E2 -14331.856} C_VEL
LIN {X 0,Y 340.772,Z 353.035,A -85,B 0,C 180,E1 -14335.664,E2 -14335.664} C_VEL
LIN {X 0,Y 340.728,Z 353.039,A -85,B 0,C 180,E1 -14338.32,E2 -14338.32} C_VEL
LIN {X 0,Y 340.696,Z 353.049,A -85,B 0,C 180,E1 -14341.044,E2 -14341.044} C_VEL
LIN {X 0,Y 340.717,Z 353.044,A -85,B 0,C 180,E1 -14345.278,E2 -14345.278} C_VEL
LIN {X 0,Y 340.717,Z 353.041,A -85,B 0,C 180,E1 -14348.387,E2 -14348.387} C_VEL
LIN {X 0,Y 340.723,Z 353.045,A -85,B 0,C 180,E1 -14351.303,E2 -14351.303} C_VEL
LIN {X 0,Y 340.817,Z 353.21,A -85,B 0,C 180,E1 -14352.816,E2 -14352.816} C_VEL
LIN {X 0,Y 341.053,Z 354.323,A -85,B 0,C 180,E1 -14353.026,E2 -14353.026} C_VEL
LIN {X 0,Y 344.736,Z 366.987,A -85,B 0,C 180,E1 -14354.211,E2 -14354.211} C_VEL
LIN {X 0,Y 346.288,Z 373.33,A -85,B 0,C 180,E1 -14354.89,E2 -14354.89} C_VEL
LIN {X 0,Y 345.511,Z 384.157,A -85,B 0,C 180,E1 -14356.064,E2 -14356.064} C_VEL
LIN {X 0,Y 344.65,Z 394.427,A -85,B 0,C 180,E1 -14357.445,E2 -14357.445} C_VEL
LIN {X 0,Y 343.662,Z 404.571,A -85,B 0,C 180,E1 -14359.125,E2 -14359.125} C_VEL
LIN {X 0,Y 342.815,Z 413.274,A -85,B 0,C 180,E1 -14360.932,E2 -14360.932} C_VEL
LIN {X 0,Y 342.212,Z 420.073,A -85,B 0,C 180,E1 -14362.687,E2 -14362.687} C_VEL
LIN {X 0,Y 341.731,Z 424.641,A -85,B 0,C 180,E1 -14364.117,E2 -14364.117} C_VEL
LIN {X 0,Y 341.308,Z 429.939,A -85,B 0,C 180,E1 -14366.223,E2 -14366.223} C_VEL
LIN {X 0,Y 341.141,Z 431.89,A -85,B 0,C 180,E1 -14367.22,E2 -14367.22} C_VEL
LIN {X 0,Y 340.354,Z 433.609,A -85,B 0,C 180,E1 -14368.162,E2 -14368.162} C_VEL
LIN {X 0,Y 337.361,Z 436.04,A -85,B 0,C 180,E1 -14369.707,E2 -14369.707} C_VEL
LIN {X 0,Y 334.492,Z 437.761,A -85,B 0,C 180,E1 -14371.301,E2 -14371.301} C_VEL
LIN {X 0,Y 333.915,Z 438.296,A -85,B 0,C 180,E1 -14372.305,E2 -14372.305} C_VEL
LIN {X 0,Y 334.044,Z 438.53,A -85,B 0,C 180,E1 -14373.78,E2 -14373.78} C_VEL
LIN {X 0,Y 334.264,Z 438.184,A -85,B 0,C 180,E1 -14375.133,E2 -14375.133} C_VEL
LIN {X 0,Y 334.859,Z 436.468,A -85,B 0,C 180,E1 -14377.435,E2 -14377.435} C_VEL
LIN {X 0,Y 335.714,Z 433.111,A -85,B 0,C 180,E1 -14379.793,E2 -14379.793} C_VEL
LIN {X 0,Y 336.619,Z 428.997,A -85,B 0,C 180,E1 -14381.749,E2 -14381.749} C_VEL
LIN {X 0,Y 337.806,Z 423.188,A -85,B 0,C 180,E1 -14383.814,E2 -14383.814} C_VEL
LIN {X 0,Y 339.073,Z 416.677,A -85,B 0,C 180,E1 -14385.598,E2 -14385.598} C_VEL
LIN {X 0,Y 340.621,Z 408.005,A -85,B 0,C 180,E1 -14387.488,E2 -14387.488} C_VEL
LIN {X 0,Y 342.029,Z 399.053,A -85,B 0,C 180,E1 -14389.043,E2 -14389.043} C_VEL
LIN {X 0,Y 343.524,Z 387.984,A -85,B 0,C 180,E1 -14390.58,E2 -14390.58} C_VEL
LIN {X 0,Y 344.086,Z 383.419,A -85,B 0,C 180,E1 -14391.114,E2 -14391.114} C_VEL
LIN {X 0,Y 343.62,Z 380.151,A -85,B 0,C 180,E1 -14391.547,E2 -14391.547} C_VEL
LIN {X 0,Y 340.201,Z 368.987,A -85,B 0,C 180,E1 -14393.055,E2 -14393.055} C_VEL
LIN {X 0,Y 335.577,Z 357.845,A -85,B 0,C 180,E1 -14394.442,E2 -14394.442} C_VEL
LIN {X 0,Y 333.976,Z 354.66,A -85,B 0,C 180,E1 -14394.869,E2 -14394.869} C_VEL
LIN {X 0,Y 333.804,Z 353.941,A -85,B 0,C 180,E1 -14395.169,E2 -14395.169} C_VEL
LIN {X 0,Y 334.095,Z 353.869,A -85,B 0,C 180,E1 -14397.589,E2 -14397.589} C_VEL
LIN {X 0,Y 334.238,Z 353.853,A -85,B 0,C 180,E1 -14400,E2 -14400} C_VEL
LIN {X 0,Y 334.095,Z 353.869,A -85,B 0,C 180,E1 -14402.411,E2 -14402.411} C_VEL
LIN {X 0,Y 333.998,Z 353.881,A -85,B 0,C 180,E1 -14406.039,E2 -14406.039} C_VEL
LIN {X 0,Y 333.812,Z 353.902,A -85,B 0,C 180,E1 -14409.697,E2 -14409.697} C_VEL
LIN {X 0,Y 333.789,Z 353.907,A -85,B 0,C 180,E1 -14413.392,E2 -14413.392} C_VEL
LIN {X 0,Y 333.711,Z 353.911,A -85,B 0,C 180,E1 -14417.148,E2 -14417.148} C_VEL
LIN {X 0,Y 333.68,Z 353.919,A -85,B 0,C 180,E1 -14419.694,E2 -14419.694} C_VEL
LIN {X 0,Y 333.662,Z 353.917,A -85,B 0,C 180,E1 -14423.591,E2 -14423.591} C_VEL
LIN {X 0,Y 333.728,Z 353.91,A -85,B 0,C 180,E1 -14426.247,E2 -14426.247} C_VEL
LIN {X 0,Y 333.684,Z 353.917,A -85,B 0,C 180,E1 -14428.975,E2 -14428.975} C_VEL
LIN {X 0,Y 333.638,Z 353.927,A -85,B 0,C 180,E1 -14432.588,E2 -14432.588} C_VEL
LIN {X 0,Y 333.669,Z 353.924,A -85,B 0,C 180,E1 -14436.14,E2 -14436.14} C_VEL
LIN {X 0,Y 333.638,Z 354.052,A -85,B 0,C 180,E1 -14440.158,E2 -14440.158} C_VEL
LIN {X 0,Y 334.89,Z 359.806,A -85,B 0,C 180,E1 -14443.832,E2 -14443.832} C_VEL
LIN {X 0,Y 336.079,Z 365.606,A -85,B 0,C 180,E1 -14447.047,E2 -14447.047} C_VEL
LIN {X 0,Y 337.379,Z 372.459,A -85,B 0,C 180,E1 -14450.422,E2 -14450.422} C_VEL
LIN {X 0,Y 337.926,Z 376.448,A -85,B 0,C 180,E1 -14452.214,E2 -14452.214} C_VEL
LIN {X 0,Y 336.269,Z 386.779,A -85,B 0,C 180,E1 -14456.287,E2 -14456.287} C_VEL
LIN {X 0,Y 335.119,Z 396.167,A -85,B 0,C 180,E1 -14459.781,E2 -14459.781} C_VEL
LIN {X 0,Y 334.077,Z 407.385,A -85,B 0,C 180,E1 -14463.783,E2 -14463.783} C_VEL
LIN {X 0,Y 333.56,Z 414.94,A -85,B 0,C 180,E1 -14466.32,E2 -14466.32} C_VEL
LIN {X 0,Y 333.998,Z 417.884,A -85,B 0,C 180,E1 -14466.557,E2 -14466.557} C_VEL
LIN {X 0,Y 336.728,Z 431.948,A -85,B 0,C 180,E1 -14467.477,E2 -14467.477} C_VEL
LIN {X 0,Y 338.071,Z 444.779,A -85,B 0,C 180,E1 -14468.427,E2 -14468.427} C_VEL
LIN {X 0,Y 338.422,Z 457.252,A -85,B 0,C 180,E1 -14469.513,E2 -14469.513} C_VEL
LIN {X 0,Y 337.9,Z 470.477,A -85,B 0,C 180,E1 -14470.878,E2 -14470.878} C_VEL
LIN {X 0,Y 337.317,Z 480.3,A -85,B 0,C 180,E1 -14472.103,E2 -14472.103} C_VEL
LIN {X 0,Y 335.711,Z 490.446,A -85,B 0,C 180,E1 -14473.584,E2 -14473.584} C_VEL
LIN {X 0,Y 334.358,Z 500.485,A -85,B 0,C 180,E1 -14475.391,E2 -14475.391} C_VEL
LIN {X 0,Y 333.773,Z 506.117,A -85,B 0,C 180,E1 -14476.608,E2 -14476.608} C_VEL
LIN {X 0,Y 332.967,Z 514.383,A -85,B 0,C 180,E1 -14478.741,E2 -14478.741} C_VEL
LIN {X 0,Y 332.592,Z 520.851,A -85,B 0,C 180,E1 -14480.881,E2 -14480.881} C_VEL
LIN {X 0,Y 332.676,Z 526.107,A -85,B 0,C 180,E1 -14483.173,E2 -14483.173} C_VEL
LIN {X 0,Y 332.944,Z 529.354,A -85,B 0,C 180,E1 -14485.157,E2 -14485.157} C_VEL
LIN {X 0,Y 333.104,Z 530.746,A -85,B 0,C 180,E1 -14486.371,E2 -14486.371} C_VEL
LIN {X 0,Y 333.548,Z 532.273,A -85,B 0,C 180,E1 -14488.793,E2 -14488.793} C_VEL
LIN {X 0,Y 333.75,Z 532.411,A -85,B 0,C 180,E1 -14490,E2 -14490} C_VEL
LIN {X 0,Y 333.559,Z 532.021,A -85,B 0,C 180,E1 -14491.207,E2 -14491.207} C_VEL
LIN {X 0,Y 333.182,Z 529.953,A -85,B 0,C 180,E1 -14493.628,E2 -14493.628} C_VEL
LIN {X 0,Y 332.997,Z 527.203,A -85,B 0,C 180,E1 -14495.45,E2 -14495.45} C_VEL
LIN {X 0,Y 332.795,Z 523.339,A -85,B 0,C 180,E1 -14497.279,E2 -14497.279} C_VEL
LIN {X 0,Y 332.73,Z 518.287,A -85,B 0,C 180,E1 -14499.115,E2 -14499.115} C_VEL
LIN {X 0,Y 332.961,Z 511.887,A -85,B 0,C 180,E1 -14500.951,E2 -14500.951} C_VEL
LIN {X 0,Y 333.509,Z 503.9,A -85,B 0,C 180,E1 -14502.783,E2 -14502.783} C_VEL
LIN {X 0,Y 334.152,Z 495.767,A -85,B 0,C 180,E1 -14504.307,E2 -14504.307} C_VEL
LIN {X 0,Y 335.213,Z 485.944,A -85,B 0,C 180,E1 -14505.816,E2 -14505.816} C_VEL
LIN {X 0,Y 336.27,Z 474.928,A -85,B 0,C 180,E1 -14507.17,E2 -14507.17} C_VEL
LIN {X 0,Y 335.976,Z 462.647,A -85,B 0,C 180,E1 -14508.409,E2 -14508.409} C_VEL
LIN {X 0,Y 335.285,Z 450.226,A -85,B 0,C 180,E1 -14509.393,E2 -14509.393} C_VEL
LIN {X 0,Y 334.251,Z 436.164,A -85,B 0,C 180,E1 -14510.239,E2 -14510.239} C_VEL
LIN {X 0,Y 333.127,Z 423.934,A -85,B 0,C 180,E1 -14510.815,E2 -14510.815} C_VEL
LIN {X 0,Y 333.596,Z 415.671,A -85,B 0,C 180,E1 -14513.595,E2 -14513.595} C_VEL
LIN {X 0,Y 334.524,Z 404.368,A -85,B 0,C 180,E1 -14517.528,E2 -14517.528} C_VEL
LIN {X 0,Y 335.69,Z 392.975,A -85,B 0,C 180,E1 -14521.56,E2 -14521.56} C_VEL
LIN {X 0,Y 337.137,Z 381.458,A -85,B 0,C 180,E1 -14525.71,E2 -14525.71} C_VEL
LIN {X 0,Y 337.848,Z 375.835,A -85,B 0,C 180,E1 -14527.769,E2 -14527.769} C_VEL
LIN {X 0,Y 336.247,Z 367.268,A -85,B 0,C 180,E1 -14531.197,E2 -14531.197} C_VEL
LIN {X 0,Y 334.472,Z 357.924,A -85,B 0,C 180,E1 -14535.133,E2 -14535.133} C_VEL
LIN {X 0,Y 333.678,Z 354,A -85,B 0,C 180,E1 -14536.893,E2 -14536.893} C_VEL
LIN {X 0,Y 333.629,Z 353.928,A -85,B 0,C 180,E1 -14541.205,E2 -14541.205} C_VEL
LIN {X 0,Y 333.669,Z 353.92,A -85,B 0,C 180,E1 -14543.86,E2 -14543.86} C_VEL
LIN {X 0,Y 333.638,Z 353.927,A -85,B 0,C 180,E1 -14547.412,E2 -14547.412} C_VEL
LIN {X 0,Y 333.704,Z 353.918,A -85,B 0,C 180,E1 -14551.027,E2 -14551.027} C_VEL
LIN {X 0,Y 333.728,Z 353.912,A -85,B 0,C 180,E1 -14553.753,E2 -14553.753} C_VEL
LIN {X 0,Y 333.649,Z 353.922,A -85,B 0,C 180,E1 -14557.719,E2 -14557.719} C_VEL
LIN {X 0,Y 333.733,Z 353.912,A -85,B 0,C 180,E1 -14561.586,E2 -14561.586} C_VEL
LIN {X 0,Y 333.801,Z 353.903,A -85,B 0,C 180,E1 -14565.576,E2 -14565.576} C_VEL
LIN {X 0,Y 333.809,Z 353.906,A -85,B 0,C 180,E1 -14569.077,E2 -14569.077} C_VEL
LIN {X 0,Y 333.983,Z 353.884,A -85,B 0,C 180,E1 -14572.747,E2 -14572.747} C_VEL
LIN {X 0,Y 333.795,Z 353.906,A -85,B 0,C 180,E1 -14575.169,E2 -14575.169} C_VEL
LIN {X 0,Y 334.095,Z 353.866,A -85,B 0,C 180,E1 -14577.589,E2 -14577.589} C_VEL
LIN {X 0,Y 334.238,Z 353.848,A -85,B 0,C 180,E1 -14580,E2 -14580} C_VEL
LIN {X 0,Y 334.095,Z 353.868,A -85,B 0,C 180,E1 -14582.411,E2 -14582.411} C_VEL
LIN {X 0,Y 333.987,Z 353.878,A -85,B 0,C 180,E1 -14586.723,E2 -14586.723} C_VEL
LIN {X 0,Y 333.853,Z 353.896,A -85,B 0,C 180,E1 -14589.695,E2 -14589.695} C_VEL
LIN {X 0,Y 333.789,Z 353.904,A -85,B 0,C 180,E1 -14593.392,E2 -14593.392} C_VEL
LIN {X 0,Y 333.739,Z 353.911,A -85,B 0,C 180,E1 -14597.147,E2 -14597.147} C_VEL
LIN {X 0,Y 333.733,Z 353.911,A -85,B 0,C 180,E1 -14599.691,E2 -14599.691} C_VEL
LIN {X 0,Y 333.686,Z 353.92,A -85,B 0,C 180,E1 -14602.279,E2 -14602.279} C_VEL
LIN {X 0,Y 333.73,Z 353.915,A -85,B 0,C 180,E1 -14606.247,E2 -14606.247} C_VEL
LIN {X 0,Y 333.705,Z 353.915,A -85,B 0,C 180,E1 -14608.973,E2 -14608.973} C_VEL
LIN {X 0,Y 333.638,Z 353.926,A -85,B 0,C 180,E1 -14612.588,E2 -14612.588} C_VEL
LIN {X 0,Y 333.671,Z 353.923,A -85,B 0,C 180,E1 -14616.14,E2 -14616.14} C_VEL
LIN {X 0,Y 333.666,Z 353.919,A -85,B 0,C 180,E1 -14619.19,E2 -14619.19} C_VEL
LIN {X 0,Y 333.657,Z 353.923,A -85,B 0,C 180,E1 -14622.506,E2 -14622.506} C_VEL
LIN {X 0,Y 333.607,Z 353.93,A -85,B 0,C 180,E1 -14625.958,E2 -14625.958} C_VEL
LIN {X 0,Y 333.645,Z 353.922,A -85,B 0,C 180,E1 -14629.316,E2 -14629.316} C_VEL
LIN {X 0,Y 333.663,Z 353.919,A -85,B 0,C 180,E1 -14633.168,E2 -14633.168} C_VEL
LIN {X 0,Y 333.64,Z 353.922,A -85,B 0,C 180,E1 -14636.793,E2 -14636.793} C_VEL
LIN {X 0,Y 333.703,Z 353.918,A -85,B 0,C 180,E1 -14639.71,E2 -14639.71} C_VEL
LIN {X 0,Y 333.744,Z 353.911,A -85,B 0,C 180,E1 -14642.402,E2 -14642.402} C_VEL
LIN {X 0,Y 333.727,Z 353.911,A -85,B 0,C 180,E1 -14645.091,E2 -14645.091} C_VEL
LIN {X 0,Y 333.682,Z 353.917,A -85,B 0,C 180,E1 -14649.02,E2 -14649.02} C_VEL
LIN {X 0,Y 333.796,Z 353.906,A -85,B 0,C 180,E1 -14651.59,E2 -14651.59} C_VEL
LIN {X 0,Y 333.81,Z 353.905,A -85,B 0,C 180,E1 -14655.577,E2 -14655.577} C_VEL
LIN {X 0,Y 333.836,Z 353.899,A -85,B 0,C 180,E1 -14659.078,E2 -14659.078} C_VEL
LIN {X 0,Y 334.028,Z 353.874,A -85,B 0,C 180,E1 -14662.748,E2 -14662.748} C_VEL
LIN {X 0,Y 333.814,Z 353.902,A -85,B 0,C 180,E1 -14665.169,E2 -14665.169} C_VEL
LIN {X 0,Y 334.134,Z 353.867,A -85,B 0,C 180,E1 -14667.589,E2 -14667.589} C_VEL
LIN {X 0,Y 334.269,Z 353.846,A -85,B 0,C 180,E1 -14670,E2 -14670} C_VEL
LIN {X 0,Y 334.11,Z 353.864,A -85,B 0,C 180,E1 -14672.411,E2 -14672.411} C_VEL
LIN {X 0,Y 334.016,Z 353.876,A -85,B 0,C 180,E1 -14676.039,E2 -14676.039} C_VEL
LIN {X 0,Y 333.861,Z 353.898,A -85,B 0,C 180,E1 -14679.695,E2 -14679.695} C_VEL
LIN {X 0,Y 333.798,Z 353.908,A -85,B 0,C 180,E1 -14683.391,E2 -14683.391} C_VEL
LIN {X 0,Y 333.748,Z 353.913,A -85,B 0,C 180,E1 -14687.146,E2 -14687.146} C_VEL
LIN {X 0,Y 333.739,Z 353.912,A -85,B 0,C 180,E1 -14689.69,E2 -14689.69} C_VEL
LIN {X 0,Y 333.693,Z 353.916,A -85,B 0,C 180,E1 -14692.278,E2 -14692.278} C_VEL
LIN {X 0,Y 333.735,Z 353.91,A -85,B 0,C 180,E1 -14696.246,E2 -14696.246} C_VEL
LIN {X 0,Y 333.689,Z 353.92,A -85,B 0,C 180,E1 -14698.973,E2 -14698.973} C_VEL
LIN {X 0,Y 333.642,Z 353.923,A -85,B 0,C 180,E1 -14702.586,E2 -14702.586} C_VEL
LIN {X 0,Y 333.676,Z 353.918,A -85,B 0,C 180,E1 -14706.138,E2 -14706.138} C_VEL
LIN {X 0,Y 333.682,Z 353.922,A -85,B 0,C 180,E1 -14709.186,E2 -14709.186} C_VEL
LIN {X 0,Y 333.764,Z 354.085,A -85,B 0,C 180,E1 -14712.499,E2 -14712.499} C_VEL
LIN {X 0,Y 333.977,Z 355.067,A -85,B 0,C 180,E1 -14712.706,E2 -14712.706} C_VEL
LIN {X 0,Y 337.594,Z 367.59,A -85,B 0,C 180,E1 -14713.895,E2 -14713.895} C_VEL
LIN {X 0,Y 339.312,Z 374.085,A -85,B 0,C 180,E1 -14714.611,E2 -14714.611} C_VEL
LIN {X 0,Y 338.532,Z 385.928,A -85,B 0,C 180,E1 -14715.935,E2 -14715.935} C_VEL
LIN {X 0,Y 337.589,Z 396.56,A -85,B 0,C 180,E1 -14717.422,E2 -14717.422} C_VEL
LIN {X 0,Y 336.669,Z 405.642,A -85,B 0,C 180,E1 -14718.973,E2 -14718.973} C_VEL
LIN {X 0,Y 335.847,Z 413.994,A -85,B 0,C 180,E1 -14720.737,E2 -14720.737} C_VEL
LIN {X 0,Y 335.217,Z 420.945,A -85,B 0,C 180,E1 -14722.555,E2 -14722.555} C_VEL
LIN {X 0,Y 334.58,Z 427.093,A -85,B 0,C 180,E1 -14724.569,E2 -14724.569} C_VEL
LIN {X 0,Y 334.165,Z 432.252,A -85,B 0,C 180,E1 -14726.851,E2 -14726.851} C_VEL
LIN {X 0,Y 333.98,Z 434.658,A -85,B 0,C 180,E1 -14728.259,E2 -14728.259} C_VEL
LIN {X 0,Y 333.879,Z 436.417,A -85,B 0,C 180,E1 -14729.656,E2 -14729.656} C_VEL
LIN {X 0,Y 333.867,Z 437.664,A -85,B 0,C 180,E1 -14731.043,E2 -14731.043} C_VEL
LIN {X 0,Y 333.915,Z 438.296,A -85,B 0,C 180,E1 -14732.305,E2 -14732.305} C_VEL
LIN {X 0,Y 333.386,Z 438.609,A -85,B 0,C 180,E1 -14733.314,E2 -14733.314} C_VEL
LIN {X 0,Y 330.792,Z 438.853,A -85,B 0,C 180,E1 -14734.967,E2 -14734.967} C_VEL
LIN {X 0,Y 328.665,Z 438.548,A -85,B 0,C 180,E1 -14736.299,E2 -14736.299} C_VEL
LIN {X 0,Y 327.909,Z 437.863,A -85,B 0,C 180,E1 -14737.316,E2 -14737.316} C_VEL
LIN {X 0,Y 327.934,Z 437.493,A -85,B 0,C 180,E1 -14737.656,E2 -14737.656} C_VEL
LIN {X 0,Y 328.574,Z 435.384,A -85,B 0,C 180,E1 -14739.334,E2 -14739.334} C_VEL
LIN {X 0,Y 329.426,Z 431.755,A -85,B 0,C 180,E1 -14741.336,E2 -14741.336} C_VEL
LIN {X 0,Y 330.711,Z 426.169,A -85,B 0,C 180,E1 -14743.556,E2 -14743.556} C_VEL
LIN {X 0,Y 332.14,Z 419.356,A -85,B 0,C 180,E1 -14745.599,E2 -14745.599} C_VEL
LIN {X 0,Y 333.457,Z 412.581,A -85,B 0,C 180,E1 -14747.215,E2 -14747.215} C_VEL
LIN {X 0,Y 334.899,Z 404.383,A -85,B 0,C 180,E1 -14748.807,E2 -14748.807} C_VEL
LIN {X 0,Y 336.487,Z 394.279,A -85,B 0,C 180,E1 -14750.381,E2 -14750.381} C_VEL
LIN {X 0,Y 337.694,Z 384.593,A -85,B 0,C 180,E1 -14751.623,E2 -14751.623} C_VEL
LIN {X 0,Y 335.002,Z 374.571,A -85,B 0,C 180,E1 -14753.072,E2 -14753.072} C_VEL
LIN {X 0,Y 331.108,Z 364.244,A -85,B 0,C 180,E1 -14754.458,E2 -14754.458} C_VEL
LIN {X 0,Y 326.906,Z 355.56,A -85,B 0,C 180,E1 -14755.646,E2 -14755.646} C_VEL
LIN {X 0,Y 326.769,Z 354.806,A -85,B 0,C 180,E1 -14755.992,E2 -14755.992} C_VEL
LIN {X 0,Y 327.036,Z 354.748,A -85,B 0,C 180,E1 -14757.537,E2 -14757.537} C_VEL
LIN {X 0,Y 327.189,Z 354.731,A -85,B 0,C 180,E1 -14760,E2 -14760} C_VEL
LIN {X 0,Y 327.036,Z 354.749,A -85,B 0,C 180,E1 -14762.463,E2 -14762.463} C_VEL
LIN {X 0,Y 326.972,Z 354.756,A -85,B 0,C 180,E1 -14766.17,E2 -14766.17} C_VEL
LIN {X 0,Y 326.775,Z 354.778,A -85,B 0,C 180,E1 -14769.908,E2 -14769.908} C_VEL
LIN {X 0,Y 326.751,Z 354.783,A -85,B 0,C 180,E1 -14773.686,E2 -14773.686} C_VEL
LIN {X 0,Y 326.656,Z 354.788,A -85,B 0,C 180,E1 -14777.53,E2 -14777.53} C_VEL
LIN {X 0,Y 326.625,Z 354.795,A -85,B 0,C 180,E1 -14780.137,E2 -14780.137} C_VEL
LIN {X 0,Y 326.642,Z 354.792,A -85,B 0,C 180,E1 -14784.13,E2 -14784.13} C_VEL
LIN {X 0,Y 326.676,Z 354.789,A -85,B 0,C 180,E1 -14786.859,E2 -14786.859} C_VEL
LIN {X 0,Y 326.628,Z 354.798,A -85,B 0,C 180,E1 -14790.61,E2 -14790.61} C_VEL
LIN {X 0,Y 326.601,Z 354.802,A -85,B 0,C 180,E1 -14794.02,E2 -14794.02} C_VEL
LIN {X 0,Y 326.618,Z 354.8,A -85,B 0,C 180,E1 -14797.238,E2 -14797.238} C_VEL
LIN {X 0,Y 326.6,Z 354.914,A -85,B 0,C 180,E1 -14799.227,E2 -14799.227} C_VEL
LIN {X 0,Y 327.645,Z 359.63,A -85,B 0,C 180,E1 -14802.462,E2 -14802.462} C_VEL
LIN {X 0,Y 328.802,Z 365.106,A -85,B 0,C 180,E1 -14805.731,E2 -14805.731} C_VEL
LIN {X 0,Y 330.134,Z 372.129,A -85,B 0,C 180,E1 -14809.413,E2 -14809.413} C_VEL
LIN {X 0,Y 330.962,Z 377.606,A -85,B 0,C 180,E1 -14811.99,E2 -14811.99} C_VEL
LIN {X 0,Y 329.775,Z 384.665,A -85,B 0,C 180,E1 -14814.873,E2 -14814.873} C_VEL
LIN {X 0,Y 328.372,Z 395.006,A -85,B 0,C 180,E1 -14818.882,E2 -14818.882} C_VEL
LIN {X 0,Y 327.327,Z 404.8,A -85,B 0,C 180,E1 -14822.509,E2 -14822.509} C_VEL
LIN {X 0,Y 326.619,Z 413.59,A -85,B 0,C 180,E1 -14825.573,E2 -14825.573} C_VEL
LIN {X 0,Y 327.218,Z 416.887,A -85,B 0,C 180,E1 -14825.845,E2 -14825.845} C_VEL
LIN {X 0,Y 329.949,Z 430.876,A -85,B 0,C 180,E1 -14826.815,E2 -14826.815} C_VEL
LIN {X 0,Y 331.356,Z 443.492,A -85,B 0,C 180,E1 -14827.803,E2 -14827.803} C_VEL
LIN {X 0,Y 331.776,Z 455.676,A -85,B 0,C 180,E1 -14828.894,E2 -14828.894} C_VEL
LIN {X 0,Y 331.309,Z 467.777,A -85,B 0,C 180,E1 -14830.16,E2 -14830.16} C_VEL
LIN {X 0,Y 330.689,Z 478.925,A -85,B 0,C 180,E1 -14831.571,E2 -14831.571} C_VEL
LIN {X 0,Y 328.881,Z 489.985,A -85,B 0,C 180,E1 -14833.233,E2 -14833.233} C_VEL
LIN {X 0,Y 327.437,Z 499.921,A -85,B 0,C 180,E1 -14835.075,E2 -14835.075} C_VEL
LIN {X 0,Y 326.62,Z 506.778,A -85,B 0,C 180,E1 -14836.626,E2 -14836.626} C_VEL
LIN {X 0,Y 325.928,Z 513.64,A -85,B 0,C 180,E1 -14838.495,E2 -14838.495} C_VEL
LIN {X 0,Y 325.536,Z 520.013,A -85,B 0,C 180,E1 -14840.682,E2 -14840.682} C_VEL
LIN {X 0,Y 325.55,Z 524.285,A -85,B 0,C 180,E1 -14842.558,E2 -14842.558} C_VEL
LIN {X 0,Y 325.686,Z 526.567,A -85,B 0,C 180,E1 -14843.806,E2 -14843.806} C_VEL
LIN {X 0,Y 325.865,Z 528.405,A -85,B 0,C 180,E1 -14845.051,E2 -14845.051} C_VEL
LIN {X 0,Y 326.053,Z 529.765,A -85,B 0,C 180,E1 -14846.293,E2 -14846.293} C_VEL
LIN {X 0,Y 326.513,Z 531.256,A -85,B 0,C 180,E1 -14848.767,E2 -14848.767} C_VEL
LIN {X 0,Y 326.736,Z 531.356,A -85,B 0,C 180,E1 -14850,E2 -14850} C_VEL
LIN {X 0,Y 326.528,Z 530.93,A -85,B 0,C 180,E1 -14851.233,E2 -14851.233} C_VEL
LIN {X 0,Y 326.136,Z 528.815,A -85,B 0,C 180,E1 -14853.707,E2 -14853.707} C_VEL
LIN {X 0,Y 325.943,Z 526.013,A -85,B 0,C 180,E1 -14855.568,E2 -14855.568} C_VEL
LIN {X 0,Y 325.742,Z 522.089,A -85,B 0,C 180,E1 -14857.438,E2 -14857.438} C_VEL
LIN {X 0,Y 325.699,Z 515.946,A -85,B 0,C 180,E1 -14859.627,E2 -14859.627} C_VEL
LIN {X 0,Y 326.043,Z 509.235,A -85,B 0,C 180,E1 -14861.501,E2 -14861.501} C_VEL
LIN {X 0,Y 326.673,Z 500.886,A -85,B 0,C 180,E1 -14863.372,E2 -14863.372} C_VEL
LIN {X 0,Y 327.579,Z 491.195,A -85,B 0,C 180,E1 -14865.105,E2 -14865.105} C_VEL
LIN {X 0,Y 328.648,Z 480.718,A -85,B 0,C 180,E1 -14866.619,E2 -14866.619} C_VEL
LIN {X 0,Y 329.219,Z 474.322,A -85,B 0,C 180,E1 -14867.389,E2 -14867.389} C_VEL
LIN {X 0,Y 328.942,Z 461.711,A -85,B 0,C 180,E1 -14868.692,E2 -14868.692} C_VEL
LIN {X 0,Y 328.22,Z 449.196,A -85,B 0,C 180,E1 -14869.706,E2 -14869.706} C_VEL
LIN {X 0,Y 327.224,Z 435.188,A -85,B 0,C 180,E1 -14870.57,E2 -14870.57} C_VEL
LIN {X 0,Y 326.077,Z 423.029,A -85,B 0,C 180,E1 -14871.162,E2 -14871.162} C_VEL
LIN {X 0,Y 326.779,Z 412.569,A -85,B 0,C 180,E1 -14874.795,E2 -14874.795} C_VEL
LIN {X 0,Y 327.791,Z 401.072,A -85,B 0,C 180,E1 -14878.92,E2 -14878.92} C_VEL
LIN {X 0,Y 328.82,Z 391.793,A -85,B 0,C 180,E1 -14882.298,E2 -14882.298} C_VEL
LIN {X 0,Y 330.419,Z 380.284,A -85,B 0,C 180,E1 -14886.551,E2 -14886.551} C_VEL
LIN {X 0,Y 330.712,Z 376.083,A -85,B 0,C 180,E1 -14888.159,E2 -14888.159} C_VEL
LIN {X 0,Y 329.093,Z 367.605,A -85,B 0,C 180,E1 -14891.63,E2 -14891.63} C_VEL
LIN {X 0,Y 327.569,Z 359.608,A -85,B 0,C 180,E1 -14895.072,E2 -14895.072} C_VEL
LIN {X 0,Y 326.612,Z 354.864,A -85,B 0,C 180,E1 -14897.283,E2 -14897.283} C_VEL
LIN {X 0,Y 326.577,Z 354.807,A -85,B 0,C 180,E1 -14901.385,E2 -14901.385} C_VEL
LIN {X 0,Y 326.613,Z 354.799,A -85,B 0,C 180,E1 -14904.851,E2 -14904.851} C_VEL
LIN {X 0,Y 326.602,Z 354.803,A -85,B 0,C 180,E1 -14907.455,E2 -14907.455} C_VEL
LIN {X 0,Y 326.655,Z 354.792,A -85,B 0,C 180,E1 -14910.34,E2 -14910.34} C_VEL
LIN {X 0,Y 326.684,Z 354.789,A -85,B 0,C 180,E1 -14914.516,E2 -14914.516} C_VEL
LIN {X 0,Y 326.611,Z 354.799,A -85,B 0,C 180,E1 -14918.543,E2 -14918.543} C_VEL
LIN {X 0,Y 326.7,Z 354.791,A -85,B 0,C 180,E1 -14921.175,E2 -14921.175} C_VEL
LIN {X 0,Y 326.756,Z 354.782,A -85,B 0,C 180,E1 -14925.433,E2 -14925.433} C_VEL
LIN {X 0,Y 326.75,Z 354.785,A -85,B 0,C 180,E1 -14928.838,E2 -14928.838} C_VEL
LIN {X 0,Y 326.933,Z 354.76,A -85,B 0,C 180,E1 -14932.589,E2 -14932.589} C_VEL
LIN {X 0,Y 326.762,Z 354.783,A -85,B 0,C 180,E1 -14935.065,E2 -14935.065} C_VEL
LIN {X 0,Y 327.036,Z 354.745,A -85,B 0,C 180,E1 -14937.537,E2 -14937.537} C_VEL
LIN {X 0,Y 327.189,Z 354.726,A -85,B 0,C 180,E1 -14940,E2 -14940} C_VEL
LIN {X 0,Y 327.035,Z 354.748,A -85,B 0,C 180,E1 -14942.463,E2 -14942.463} C_VEL
LIN {X 0,Y 326.952,Z 354.754,A -85,B 0,C 180,E1 -14946.717,E2 -14946.717} C_VEL
LIN {X 0,Y 326.804,Z 354.774,A -85,B 0,C 180,E1 -14949.907,E2 -14949.907} C_VEL
LIN {X 0,Y 326.751,Z 354.78,A -85,B 0,C 180,E1 -14953.686,E2 -14953.686} C_VEL
LIN {X 0,Y 326.692,Z 354.788,A -85,B 0,C 180,E1 -14957.528,E2 -14957.528} C_VEL
LIN {X 0,Y 326.658,Z 354.794,A -85,B 0,C 180,E1 -14960.135,E2 -14960.135} C_VEL
LIN {X 0,Y 326.645,Z 354.796,A -85,B 0,C 180,E1 -14964.129,E2 -14964.129} C_VEL
LIN {X 0,Y 326.679,Z 354.791,A -85,B 0,C 180,E1 -14966.858,E2 -14966.858} C_VEL
LIN {X 0,Y 326.633,Z 354.798,A -85,B 0,C 180,E1 -14970.612,E2 -14970.612} C_VEL
LIN {X 0,Y 326.601,Z 354.802,A -85,B 0,C 180,E1 -14974.02,E2 -14974.02} C_VEL
LIN {X 0,Y 326.624,Z 354.796,A -85,B 0,C 180,E1 -14977.239,E2 -14977.239} C_VEL
LIN {X 0,Y 326.599,Z 354.805,A -85,B 0,C 180,E1 -14980.208,E2 -14980.208} C_VEL
LIN {X 0,Y 326.574,Z 354.803,A -85,B 0,C 180,E1 -14983.524,E2 -14983.524} C_VEL
LIN {X 0,Y 326.578,Z 354.802,A -85,B 0,C 180,E1 -14987.028,E2 -14987.028} C_VEL
LIN {X 0,Y 326.609,Z 354.798,A -85,B 0,C 180,E1 -14990.773,E2 -14990.773} C_VEL
LIN {X 0,Y 326.611,Z 354.8,A -85,B 0,C 180,E1 -14994.481,E2 -14994.481} C_VEL
LIN {X 0,Y 326.614,Z 354.799,A -85,B 0,C 180,E1 -14997.457,E2 -14997.457} C_VEL
LIN {X 0,Y 326.661,Z 354.794,A -85,B 0,C 180,E1 -15000.342,E2 -15000.342} C_VEL
LIN {X 0,Y 326.685,Z 354.789,A -85,B 0,C 180,E1 -15003.143,E2 -15003.143} C_VEL
LIN {X 0,Y 326.652,Z 354.798,A -85,B 0,C 180,E1 -15005.872,E2 -15005.872} C_VEL
LIN {X 0,Y 326.666,Z 354.796,A -85,B 0,C 180,E1 -15009.866,E2 -15009.866} C_VEL
LIN {X 0,Y 326.701,Z 354.787,A -85,B 0,C 180,E1 -15012.473,E2 -15012.473} C_VEL
LIN {X 0,Y 326.761,Z 354.78,A -85,B 0,C 180,E1 -15016.315,E2 -15016.315} C_VEL
LIN {X 0,Y 326.816,Z 354.774,A -85,B 0,C 180,E1 -15020.094,E2 -15020.094} C_VEL
LIN {X 0,Y 326.982,Z 354.752,A -85,B 0,C 180,E1 -15022.591,E2 -15022.591} C_VEL
LIN {X 0,Y 326.781,Z 354.778,A -85,B 0,C 180,E1 -15025.065,E2 -15025.065} C_VEL
LIN {X 0,Y 327.07,Z 354.746,A -85,B 0,C 180,E1 -15027.537,E2 -15027.537} C_VEL
LIN {X 0,Y 327.219,Z 354.724,A -85,B 0,C 180,E1 -15030,E2 -15030} C_VEL
LIN {X 0,Y 327.051,Z 354.743,A -85,B 0,C 180,E1 -15032.463,E2 -15032.463} C_VEL
LIN {X 0,Y 326.991,Z 354.751,A -85,B 0,C 180,E1 -15036.169,E2 -15036.169} C_VEL
LIN {X 0,Y 326.813,Z 354.774,A -85,B 0,C 180,E1 -15039.906,E2 -15039.906} C_VEL
LIN {X 0,Y 326.76,Z 354.782,A -85,B 0,C 180,E1 -15043.685,E2 -15043.685} C_VEL
LIN {X 0,Y 326.7,Z 354.79,A -85,B 0,C 180,E1 -15047.527,E2 -15047.527} C_VEL
LIN {X 0,Y 326.666,Z 354.791,A -85,B 0,C 180,E1 -15050.134,E2 -15050.134} C_VEL
LIN {X 0,Y 326.652,Z 354.793,A -85,B 0,C 180,E1 -15054.128,E2 -15054.128} C_VEL
LIN {X 0,Y 326.682,Z 354.792,A -85,B 0,C 180,E1 -15056.857,E2 -15056.857} C_VEL
LIN {X 0,Y 326.633,Z 354.796,A -85,B 0,C 180,E1 -15060.609,E2 -15060.609} C_VEL
LIN {X 0,Y 326.605,Z 354.798,A -85,B 0,C 180,E1 -15064.019,E2 -15064.019} C_VEL
LIN {X 0,Y 326.629,Z 354.799,A -85,B 0,C 180,E1 -15067.239,E2 -15067.239} C_VEL
LIN {X 0,Y 326.664,Z 354.796,A -85,B 0,C 180,E1 -15071.148,E2 -15071.148} C_VEL
LIN {X 0,Y 326.708,Z 354.97,A -85,B 0,C 180,E1 -15072.187,E2 -15072.187} C_VEL
LIN {X 0,Y 326.986,Z 356.104,A -85,B 0,C 180,E1 -15072.402,E2 -15072.402} C_VEL
LIN {X 0,Y 330.6,Z 368.652,A -85,B 0,C 180,E1 -15073.616,E2 -15073.616} C_VEL
LIN {X 0,Y 332.406,Z 375.468,A -85,B 0,C 180,E1 -15074.389,E2 -15074.389} C_VEL
LIN {X 0,Y 331.689,Z 386.4,A -85,B 0,C 180,E1 -15075.635,E2 -15075.635} C_VEL
LIN {X 0,Y 330.699,Z 397.121,A -85,B 0,C 180,E1 -15077.151,E2 -15077.151} C_VEL
LIN {X 0,Y 329.784,Z 405.831,A -85,B 0,C 180,E1 -15078.651,E2 -15078.651} C_VEL
LIN {X 0,Y 328.868,Z 414.871,A -85,B 0,C 180,E1 -15080.574,E2 -15080.574} C_VEL
LIN {X 0,Y 328.249,Z 421.702,A -85,B 0,C 180,E1 -15082.389,E2 -15082.389} C_VEL
LIN {X 0,Y 327.539,Z 428.303,A -85,B 0,C 180,E1 -15084.596,E2 -15084.596} C_VEL
LIN {X 0,Y 327.116,Z 433.395,A -85,B 0,C 180,E1 -15086.917,E2 -15086.917} C_VEL
LIN {X 0,Y 326.895,Z 436.545,A -85,B 0,C 180,E1 -15088.937,E2 -15088.937} C_VEL
LIN {X 0,Y 326.837,Z 438.084,A -85,B 0,C 180,E1 -15090.358,E2 -15090.358} C_VEL
LIN {X 0,Y 326.881,Z 439.26,A -85,B 0,C 180,E1 -15092.307,E2 -15092.307} C_VEL
LIN {X 0,Y 327.149,Z 439.501,A -85,B 0,C 180,E1 -15094.455,E2 -15094.455} C_VEL
LIN {X 0,Y 327.453,Z 438.961,A -85,B 0,C 180,E1 -15095.934,E2 -15095.934} C_VEL
LIN {X 0,Y 327.934,Z 437.493,A -85,B 0,C 180,E1 -15097.656,E2 -15097.656} C_VEL
LIN {X 0,Y 327.632,Z 436.486,A -85,B 0,C 180,E1 -15098.668,E2 -15098.668} C_VEL
LIN {X 0,Y 325.487,Z 434.541,A -85,B 0,C 180,E1 -15100.332,E2 -15100.332} C_VEL
LIN {X 0,Y 323.48,Z 432,A -85,B 0,C 180,E1 -15101.987,E2 -15101.987} C_VEL
LIN {X 0,Y 323.4,Z 429.861,A -85,B 0,C 180,E1 -15102.968,E2 -15102.968} C_VEL
LIN {X 0,Y 324.747,Z 424.148,A -85,B 0,C 180,E1 -15104.948,E2 -15104.948} C_VEL
LIN {X 0,Y 326.276,Z 416.878,A -85,B 0,C 180,E1 -15106.928,E2 -15106.928} C_VEL
LIN {X 0,Y 327.748,Z 409.384,A -85,B 0,C 180,E1 -15108.559,E2 -15108.559} C_VEL
LIN {X 0,Y 329.369,Z 400.245,A -85,B 0,C 180,E1 -15110.171,E2 -15110.171} C_VEL
LIN {X 0,Y 330.881,Z 390.261,A -85,B 0,C 180,E1 -15111.603,E2 -15111.603} C_VEL
LIN {X 0,Y 331.306,Z 386.51,A -85,B 0,C 180,E1 -15112.072,E2 -15112.072} C_VEL
LIN {X 0,Y 328.639,Z 376.761,A -85,B 0,C 180,E1 -15113.554,E2 -15113.554} C_VEL
LIN {X 0,Y 325.229,Z 367.529,A -85,B 0,C 180,E1 -15114.886,E2 -15114.886} C_VEL
LIN {X 0,Y 319.915,Z 356.442,A -85,B 0,C 180,E1 -15116.458,E2 -15116.458} C_VEL
LIN {X 0,Y 319.822,Z 355.683,A -85,B 0,C 180,E1 -15116.772,E2 -15116.772} C_VEL
LIN {X 0,Y 320.141,Z 355.608,A -85,B 0,C 180,E1 -15120,E2 -15120} C_VEL
LIN {X 0,Y 319.98,Z 355.628,A -85,B 0,C 180,E1 -15122.518,E2 -15122.518} C_VEL
LIN {X 0,Y 319.926,Z 355.633,A -85,B 0,C 180,E1 -15126.306,E2 -15126.306} C_VEL
LIN {X 0,Y 319.727,Z 355.656,A -85,B 0,C 180,E1 -15130.128,E2 -15130.128} C_VEL
LIN {X 0,Y 319.724,Z 355.659,A -85,B 0,C 180,E1 -15133.993,E2 -15133.993} C_VEL
LIN {X 0,Y 319.617,Z 355.665,A -85,B 0,C 180,E1 -15137.929,E2 -15137.929} C_VEL
LIN {X 0,Y 319.561,Z 355.68,A -85,B 0,C 180,E1 -15141.955,E2 -15141.955} C_VEL
LIN {X 0,Y 319.612,Z 355.668,A -85,B 0,C 180,E1 -15146.09,E2 -15146.09} C_VEL
LIN {X 0,Y 319.574,Z 355.674,A -85,B 0,C 180,E1 -15148.935,E2 -15148.935} C_VEL
LIN {X 0,Y 319.524,Z 355.683,A -85,B 0,C 180,E1 -15151.863,E2 -15151.863} C_VEL
LIN {X 0,Y 319.574,Z 355.676,A -85,B 0,C 180,E1 -15155.543,E2 -15155.543} C_VEL
LIN {X 0,Y 319.549,Z 355.779,A -85,B 0,C 180,E1 -15158.212,E2 -15158.212} C_VEL
LIN {X 0,Y 320.625,Z 360.744,A -85,B 0,C 180,E1 -15161.819,E2 -15161.819} C_VEL
LIN {X 0,Y 321.964,Z 367.003,A -85,B 0,C 180,E1 -15165.694,E2 -15165.694} C_VEL
LIN {X 0,Y 323.323,Z 374.191,A -85,B 0,C 180,E1 -15169.534,E2 -15169.534} C_VEL
LIN {X 0,Y 323.931,Z 377.94,A -85,B 0,C 180,E1 -15171.358,E2 -15171.358} C_VEL
LIN {X 0,Y 323.821,Z 380.653,A -85,B 0,C 180,E1 -15172.578,E2 -15172.578} C_VEL
LIN {X 0,Y 322.009,Z 391.31,A -85,B 0,C 180,E1 -15176.933,E2 -15176.933} C_VEL
LIN {X 0,Y 320.622,Z 402.498,A -85,B 0,C 180,E1 -15181.259,E2 -15181.259} C_VEL
LIN {X 0,Y 319.721,Z 412.094,A -85,B 0,C 180,E1 -15184.749,E2 -15184.749} C_VEL
LIN {X 0,Y 319.785,Z 413.131,A -85,B 0,C 180,E1 -15184.885,E2 -15184.885} C_VEL
LIN {X 0,Y 322.946,Z 428.302,A -85,B 0,C 180,E1 -15185.995,E2 -15185.995} C_VEL
LIN {X 0,Y 324.669,Z 441.44,A -85,B 0,C 180,E1 -15187.068,E2 -15187.068} C_VEL
LIN {X 0,Y 325.156,Z 453.129,A -85,B 0,C 180,E1 -15188.143,E2 -15188.143} C_VEL
LIN {X 0,Y 324.69,Z 466.723,A -85,B 0,C 180,E1 -15189.601,E2 -15189.601} C_VEL
LIN {X 0,Y 323.982,Z 477.649,A -85,B 0,C 180,E1 -15191.011,E2 -15191.011} C_VEL
LIN {X 0,Y 322.371,Z 487.814,A -85,B 0,C 180,E1 -15192.557,E2 -15192.557} C_VEL
LIN {X 0,Y 320.765,Z 497.86,A -85,B 0,C 180,E1 -15194.431,E2 -15194.431} C_VEL
LIN {X 0,Y 319.688,Z 506.121,A -85,B 0,C 180,E1 -15196.33,E2 -15196.33} C_VEL
LIN {X 0,Y 318.797,Z 513.878,A -85,B 0,C 180,E1 -15198.556,E2 -15198.556} C_VEL
LIN {X 0,Y 318.452,Z 519.198,A -85,B 0,C 180,E1 -15200.473,E2 -15200.473} C_VEL
LIN {X 0,Y 318.468,Z 523.41,A -85,B 0,C 180,E1 -15202.391,E2 -15202.391} C_VEL
LIN {X 0,Y 318.62,Z 525.666,A -85,B 0,C 180,E1 -15203.668,E2 -15203.668} C_VEL
LIN {X 0,Y 318.791,Z 527.447,A -85,B 0,C 180,E1 -15204.941,E2 -15204.941} C_VEL
LIN {X 0,Y 319.001,Z 528.79,A -85,B 0,C 180,E1 -15206.21,E2 -15206.21} C_VEL
LIN {X 0,Y 319.478,Z 530.24,A -85,B 0,C 180,E1 -15208.74,E2 -15208.74} C_VEL
LIN {X 0,Y 319.719,Z 530.291,A -85,B 0,C 180,E1 -15210,E2 -15210} C_VEL
LIN {X 0,Y 319.497,Z 529.84,A -85,B 0,C 180,E1 -15211.26,E2 -15211.26} C_VEL
LIN {X 0,Y 319.19,Z 528.956,A -85,B 0,C 180,E1 -15212.524,E2 -15212.524} C_VEL
LIN {X 0,Y 319.089,Z 527.658,A -85,B 0,C 180,E1 -15213.789,E2 -15213.789} C_VEL
LIN {X 0,Y 318.892,Z 524.799,A -85,B 0,C 180,E1 -15215.692,E2 -15215.692} C_VEL
LIN {X 0,Y 318.683,Z 520.802,A -85,B 0,C 180,E1 -15217.603,E2 -15217.603} C_VEL
LIN {X 0,Y 318.67,Z 514.573,A -85,B 0,C 180,E1 -15219.841,E2 -15219.841} C_VEL
LIN {X 0,Y 319.042,Z 507.784,A -85,B 0,C 180,E1 -15221.757,E2 -15221.757} C_VEL
LIN {X 0,Y 319.689,Z 499.286,A -85,B 0,C 180,E1 -15223.669,E2 -15223.669} C_VEL
LIN {X 0,Y 320.569,Z 490.436,A -85,B 0,C 180,E1 -15225.282,E2 -15225.282} C_VEL
LIN {X 0,Y 321.672,Z 480.033,A -85,B 0,C 180,E1 -15226.827,E2 -15226.827} C_VEL
LIN {X 0,Y 322.16,Z 473.659,A -85,B 0,C 180,E1 -15227.619,E2 -15227.619} C_VEL
LIN {X 0,Y 321.869,Z 461.121,A -85,B 0,C 180,E1 -15228.953,E2 -15228.953} C_VEL
LIN {X 0,Y 321.256,Z 449.652,A -85,B 0,C 180,E1 -15229.927,E2 -15229.927} C_VEL
LIN {X 0,Y 320.256,Z 435.42,A -85,B 0,C 180,E1 -15230.849,E2 -15230.849} C_VEL
LIN {X 0,Y 319.046,Z 422.132,A -85,B 0,C 180,E1 -15231.524,E2 -15231.524} C_VEL
LIN {X 0,Y 319.503,Z 415.071,A -85,B 0,C 180,E1 -15234.012,E2 -15234.012} C_VEL
LIN {X 0,Y 320.478,Z 403.917,A -85,B 0,C 180,E1 -15238.094,E2 -15238.094} C_VEL
LIN {X 0,Y 321.781,Z 392.49,A -85,B 0,C 180,E1 -15242.35,E2 -15242.35} C_VEL
LIN {X 0,Y 323.502,Z 380.523,A -85,B 0,C 180,E1 -15246.887,E2 -15246.887} C_VEL
LIN {X 0,Y 323.743,Z 377.713,A -85,B 0,C 180,E1 -15247.976,E2 -15247.976} C_VEL
LIN {X 0,Y 322.539,Z 370.887,A -85,B 0,C 180,E1 -15250.819,E2 -15250.819} C_VEL
LIN {X 0,Y 320.888,Z 362.44,A -85,B 0,C 180,E1 -15254.494,E2 -15254.494} C_VEL
LIN {X 0,Y 319.595,Z 355.752,A -85,B 0,C 180,E1 -15257.59,E2 -15257.59} C_VEL
LIN {X 0,Y 319.54,Z 355.679,A -85,B 0,C 180,E1 -15260.37,E2 -15260.37} C_VEL
LIN {X 0,Y 319.574,Z 355.675,A -85,B 0,C 180,E1 -15264.457,E2 -15264.457} C_VEL
LIN {X 0,Y 319.527,Z 355.68,A -85,B 0,C 180,E1 -15268.137,E2 -15268.137} C_VEL
LIN {X 0,Y 319.61,Z 355.672,A -85,B 0,C 180,E1 -15271.588,E2 -15271.588} C_VEL
LIN {X 0,Y 319.597,Z 355.676,A -85,B 0,C 180,E1 -15275.303,E2 -15275.303} C_VEL
LIN {X 0,Y 319.579,Z 355.677,A -85,B 0,C 180,E1 -15279.399,E2 -15279.399} C_VEL
LIN {X 0,Y 319.617,Z 355.669,A -85,B 0,C 180,E1 -15282.071,E2 -15282.071} C_VEL
LIN {X 0,Y 319.724,Z 355.655,A -85,B 0,C 180,E1 -15286.007,E2 -15286.007} C_VEL
LIN {X 0,Y 319.727,Z 355.655,A -85,B 0,C 180,E1 -15289.872,E2 -15289.872} C_VEL
LIN {X 0,Y 319.911,Z 355.633,A -85,B 0,C 180,E1 -15293.694,E2 -15293.694} C_VEL
LIN {X 0,Y 319.979,Z 355.624,A -85,B 0,C 180,E1 -15297.482,E2 -15297.482} C_VEL
LIN {X 0,Y 320.141,Z 355.604,A -85,B 0,C 180,E1 -15300,E2 -15300} C_VEL
LIN {X 0,Y 319.979,Z 355.627,A -85,B 0,C 180,E1 -15302.518,E2 -15302.518} C_VEL
LIN {X 0,Y 319.914,Z 355.631,A -85,B 0,C 180,E1 -15306.709,E2 -15306.709} C_VEL
LIN {X 0,Y 319.749,Z 355.654,A -85,B 0,C 180,E1 -15310.127,E2 -15310.127} C_VEL
LIN {X 0,Y 319.724,Z 355.66,A -85,B 0,C 180,E1 -15314.724,E2 -15314.724} C_VEL
LIN {X 0,Y 319.683,Z 355.662,A -85,B 0,C 180,E1 -15319.038,E2 -15319.038} C_VEL
LIN {X 0,Y 319.564,Z 355.676,A -85,B 0,C 180,E1 -15323.32,E2 -15323.32} C_VEL
LIN {X 0,Y 319.629,Z 355.67,A -85,B 0,C 180,E1 -15326.089,E2 -15326.089} C_VEL
LIN {X 0,Y 319.584,Z 355.674,A -85,B 0,C 180,E1 -15328.934,E2 -15328.934} C_VEL
LIN {X 0,Y 319.526,Z 355.682,A -85,B 0,C 180,E1 -15331.862,E2 -15331.862} C_VEL
LIN {X 0,Y 319.575,Z 355.675,A -85,B 0,C 180,E1 -15335.544,E2 -15335.544} C_VEL
LIN {X 0,Y 319.576,Z 355.677,A -85,B 0,C 180,E1 -15338.008,E2 -15338.008} C_VEL
LIN {X 0,Y 319.562,Z 355.677,A -85,B 0,C 180,E1 -15341.606,E2 -15341.606} C_VEL
LIN {X 0,Y 319.498,Z 355.684,A -85,B 0,C 180,E1 -15345.26,E2 -15345.26} C_VEL
LIN {X 0,Y 319.527,Z 355.681,A -85,B 0,C 180,E1 -15348.713,E2 -15348.713} C_VEL
LIN {X 0,Y 319.575,Z 355.677,A -85,B 0,C 180,E1 -15352.345,E2 -15352.345} C_VEL
LIN {X 0,Y 319.559,Z 355.676,A -85,B 0,C 180,E1 -15355.124,E2 -15355.124} C_VEL
LIN {X 0,Y 319.573,Z 355.674,A -85,B 0,C 180,E1 -15359.057,E2 -15359.057} C_VEL
LIN {X 0,Y 319.617,Z 355.67,A -85,B 0,C 180,E1 -15362.5,E2 -15362.5} C_VEL
LIN {X 0,Y 319.605,Z 355.671,A -85,B 0,C 180,E1 -15365.305,E2 -15365.305} C_VEL
LIN {X 0,Y 319.597,Z 355.675,A -85,B 0,C 180,E1 -15368.048,E2 -15368.048} C_VEL
LIN {X 0,Y 319.69,Z 355.66,A -85,B 0,C 180,E1 -15370.962,E2 -15370.962} C_VEL
LIN {X 0,Y 319.732,Z 355.656,A -85,B 0,C 180,E1 -15375.276,E2 -15375.276} C_VEL
LIN {X 0,Y 319.76,Z 355.655,A -85,B 0,C 180,E1 -15379.873,E2 -15379.873} C_VEL
LIN {X 0,Y 319.936,Z 355.63,A -85,B 0,C 180,E1 -15382.426,E2 -15382.426} C_VEL
LIN {X 0,Y 319.751,Z 355.653,A -85,B 0,C 180,E1 -15384.956,E2 -15384.956} C_VEL
LIN {X 0,Y 320.011,Z 355.625,A -85,B 0,C 180,E1 -15387.483,E2 -15387.483} C_VEL
LIN {X 0,Y 320.171,Z 355.602,A -85,B 0,C 180,E1 -15390,E2 -15390} C_VEL
LIN {X 0,Y 319.994,Z 355.622,A -85,B 0,C 180,E1 -15392.518,E2 -15392.518} C_VEL
LIN {X 0,Y 319.945,Z 355.628,A -85,B 0,C 180,E1 -15396.305,E2 -15396.305} C_VEL
LIN {X 0,Y 319.839,Z 355.642,A -85,B 0,C 180,E1 -15398.848,E2 -15398.848} C_VEL
LIN {X 0,Y 319.683,Z 355.661,A -85,B 0,C 180,E1 -15402.699,E2 -15402.699} C_VEL
LIN {X 0,Y 319.701,Z 355.664,A -85,B 0,C 180,E1 -15405.295,E2 -15405.295} C_VEL
LIN {X 0,Y 319.675,Z 355.667,A -85,B 0,C 180,E1 -15409.254,E2 -15409.254} C_VEL
LIN {X 0,Y 319.57,Z 355.68,A -85,B 0,C 180,E1 -15413.319,E2 -15413.319} C_VEL
LIN {X 0,Y 319.618,Z 355.669,A -85,B 0,C 180,E1 -15416.089,E2 -15416.089} C_VEL
LIN {X 0,Y 319.579,Z 355.677,A -85,B 0,C 180,E1 -15418.934,E2 -15418.934} C_VEL
LIN {X 0,Y 319.529,Z 355.68,A -85,B 0,C 180,E1 -15421.861,E2 -15421.861} C_VEL
LIN {X 0,Y 319.579,Z 355.675,A -85,B 0,C 180,E1 -15425.542,E2 -15425.542} C_VEL
LIN {X 0,Y 319.598,Z 355.672,A -85,B 0,C 180,E1 -15428.003,E2 -15428.003} C_VEL
LIN {X 0,Y 319.637,Z 355.817,A -85,B 0,C 180,E1 -15431.845,E2 -15431.845} C_VEL
LIN {X 0,Y 319.902,Z 356.947,A -85,B 0,C 180,E1 -15432.072,E2 -15432.072} C_VEL
LIN {X 0,Y 323.463,Z 369.171,A -85,B 0,C 180,E1 -15433.285,E2 -15433.285} C_VEL
LIN {X 0,Y 325.574,Z 377.167,A -85,B 0,C 180,E1 -15434.209,E2 -15434.209} C_VEL
LIN {X 0,Y 324.668,Z 388.745,A -85,B 0,C 180,E1 -15435.588,E2 -15435.588} C_VEL
LIN {X 0,Y 323.574,Z 399.978,A -85,B 0,C 180,E1 -15437.254,E2 -15437.254} C_VEL
LIN {X 0,Y 322.7,Z 408.368,A -85,B 0,C 180,E1 -15438.791,E2 -15438.791} C_VEL
LIN {X 0,Y 321.764,Z 416.858,A -85,B 0,C 180,E1 -15440.697,E2 -15440.697} C_VEL
LIN {X 0,Y 321.089,Z 423.695,A -85,B 0,C 180,E1 -15442.599,E2 -15442.599} C_VEL
LIN {X 0,Y 320.483,Z 429.697,A -85,B 0,C 180,E1 -15444.716,E2 -15444.716} C_VEL
LIN {X 0,Y 320.11,Z 434.021,A -85,B 0,C 180,E1 -15446.71,E2 -15446.71} C_VEL
LIN {X 0,Y 319.854,Z 437.559,A -85,B 0,C 180,E1 -15448.971,E2 -15448.971} C_VEL
LIN {X 0,Y 319.832,Z 439.911,A -85,B 0,C 180,E1 -15451.515,E2 -15451.515} C_VEL
LIN {X 0,Y 320.044,Z 440.642,A -85,B 0,C 180,E1 -15453.948,E2 -15453.948} C_VEL
LIN {X 0,Y 320.302,Z 440.377,A -85,B 0,C 180,E1 -15455.361,E2 -15455.361} C_VEL
LIN {X 0,Y 320.992,Z 438.729,A -85,B 0,C 180,E1 -15457.768,E2 -15457.768} C_VEL
LIN {X 0,Y 321.802,Z 436.079,A -85,B 0,C 180,E1 -15459.897,E2 -15459.897} C_VEL
LIN {X 0,Y 322.583,Z 433.023,A -85,B 0,C 180,E1 -15461.584,E2 -15461.584} C_VEL
LIN {X 0,Y 323.4,Z 429.861,A -85,B 0,C 180,E1 -15462.968,E2 -15462.968} C_VEL
LIN {X 0,Y 323.387,Z 427.57,A -85,B 0,C 180,E1 -15463.933,E2 -15463.933} C_VEL
LIN {X 0,Y 321.754,Z 423.617,A -85,B 0,C 180,E1 -15465.521,E2 -15465.521} C_VEL
LIN {X 0,Y 320.183,Z 419.023,A -85,B 0,C 180,E1 -15467.061,E2 -15467.061} C_VEL
LIN {X 0,Y 320.255,Z 415.698,A -85,B 0,C 180,E1 -15467.936,E2 -15467.936} C_VEL
LIN {X 0,Y 321.985,Z 407.106,A -85,B 0,C 180,E1 -15469.714,E2 -15469.714} C_VEL
LIN {X 0,Y 323.841,Z 396.665,A -85,B 0,C 180,E1 -15471.419,E2 -15471.419} C_VEL
LIN {X 0,Y 324.911,Z 389.538,A -85,B 0,C 180,E1 -15472.387,E2 -15472.387} C_VEL
LIN {X 0,Y 323.244,Z 381.916,A -85,B 0,C 180,E1 -15473.607,E2 -15473.607} C_VEL
LIN {X 0,Y 320.02,Z 372.511,A -85,B 0,C 180,E1 -15475.059,E2 -15475.059} C_VEL
LIN {X 0,Y 314.161,Z 359.903,A -85,B 0,C 180,E1 -15476.954,E2 -15476.954} C_VEL
LIN {X 0,Y 313.03,Z 357.253,A -85,B 0,C 180,E1 -15477.346,E2 -15477.346} C_VEL
LIN {X 0,Y 312.944,Z 356.536,A -85,B 0,C 180,E1 -15477.667,E2 -15477.667} C_VEL
LIN {X 0,Y 313.094,Z 356.486,A -85,B 0,C 180,E1 -15480,E2 -15480} C_VEL
LIN {X 0,Y 312.926,Z 356.507,A -85,B 0,C 180,E1 -15482.575,E2 -15482.575} C_VEL
LIN {X 0,Y 312.883,Z 356.51,A -85,B 0,C 180,E1 -15486.449,E2 -15486.449} C_VEL
LIN {X 0,Y 312.677,Z 356.535,A -85,B 0,C 180,E1 -15490.359,E2 -15490.359} C_VEL
LIN {X 0,Y 312.66,Z 356.54,A -85,B 0,C 180,E1 -15494.865,E2 -15494.865} C_VEL
LIN {X 0,Y 312.579,Z 356.551,A -85,B 0,C 180,E1 -15499.213,E2 -15499.213} C_VEL
LIN {X 0,Y 312.519,Z 356.554,A -85,B 0,C 180,E1 -15502.781,E2 -15502.781} C_VEL
LIN {X 0,Y 312.59,Z 356.543,A -85,B 0,C 180,E1 -15505.934,E2 -15505.934} C_VEL
LIN {X 0,Y 312.532,Z 356.554,A -85,B 0,C 180,E1 -15509.651,E2 -15509.651} C_VEL
LIN {X 0,Y 312.514,Z 356.555,A -85,B 0,C 180,E1 -15513.689,E2 -15513.689} C_VEL
LIN {X 0,Y 312.519,Z 356.722,A -85,B 0,C 180,E1 -15517.191,E2 -15517.191} C_VEL
LIN {X 0,Y 313.44,Z 361.059,A -85,B 0,C 180,E1 -15520.56,E2 -15520.56} C_VEL
LIN {X 0,Y 314.515,Z 365.919,A -85,B 0,C 180,E1 -15523.845,E2 -15523.845} C_VEL
LIN {X 0,Y 315.67,Z 371.786,A -85,B 0,C 180,E1 -15527.283,E2 -15527.283} C_VEL
LIN {X 0,Y 316.944,Z 378.695,A -85,B 0,C 180,E1 -15530.905,E2 -15530.905} C_VEL
LIN {X 0,Y 316.912,Z 381.98,A -85,B 0,C 180,E1 -15532.423,E2 -15532.423} C_VEL
LIN {X 0,Y 315.019,Z 392.565,A -85,B 0,C 180,E1 -15536.868,E2 -15536.868} C_VEL
LIN {X 0,Y 313.694,Z 402.701,A -85,B 0,C 180,E1 -15540.898,E2 -15540.898} C_VEL
LIN {X 0,Y 312.895,Z 410.74,A -85,B 0,C 180,E1 -15543.892,E2 -15543.892} C_VEL
LIN {X 0,Y 313.387,Z 413.727,A -85,B 0,C 180,E1 -15544.18,E2 -15544.18} C_VEL
LIN {X 0,Y 315.872,Z 425.114,A -85,B 0,C 180,E1 -15545.063,E2 -15545.063} C_VEL
LIN {X 0,Y 317.937,Z 439.815,A -85,B 0,C 180,E1 -15546.323,E2 -15546.323} C_VEL
LIN {X 0,Y 318.557,Z 451.78,A -85,B 0,C 180,E1 -15547.461,E2 -15547.461} C_VEL
LIN {X 0,Y 318.241,Z 463.719,A -85,B 0,C 180,E1 -15548.771,E2 -15548.771} C_VEL
LIN {X 0,Y 317.31,Z 475.229,A -85,B 0,C 180,E1 -15550.26,E2 -15550.26} C_VEL
LIN {X 0,Y 316.653,Z 481.718,A -85,B 0,C 180,E1 -15551.227,E2 -15551.227} C_VEL
LIN {X 0,Y 314.669,Z 492.687,A -85,B 0,C 180,E1 -15553.122,E2 -15553.122} C_VEL
LIN {X 0,Y 313.308,Z 500.901,A -85,B 0,C 180,E1 -15554.867,E2 -15554.867} C_VEL
LIN {X 0,Y 312.534,Z 506.694,A -85,B 0,C 180,E1 -15556.343,E2 -15556.343} C_VEL
LIN {X 0,Y 311.78,Z 513.145,A -85,B 0,C 180,E1 -15558.295,E2 -15558.295} C_VEL
LIN {X 0,Y 311.378,Z 518.392,A -85,B 0,C 180,E1 -15560.254,E2 -15560.254} C_VEL
LIN {X 0,Y 311.369,Z 522.544,A -85,B 0,C 180,E1 -15562.217,E2 -15562.217} C_VEL
LIN {X 0,Y 311.528,Z 524.764,A -85,B 0,C 180,E1 -15563.523,E2 -15563.523} C_VEL
LIN {X 0,Y 311.701,Z 526.496,A -85,B 0,C 180,E1 -15564.826,E2 -15564.826} C_VEL
LIN {X 0,Y 311.948,Z 527.817,A -85,B 0,C 180,E1 -15566.125,E2 -15566.125} C_VEL
LIN {X 0,Y 312.044,Z 528.707,A -85,B 0,C 180,E1 -15567.418,E2 -15567.418} C_VEL
LIN {X 0,Y 312.441,Z 529.207,A -85,B 0,C 180,E1 -15568.711,E2 -15568.711} C_VEL
LIN {X 0,Y 312.701,Z 529.227,A -85,B 0,C 180,E1 -15570,E2 -15570} C_VEL
LIN {X 0,Y 312.465,Z 528.753,A -85,B 0,C 180,E1 -15571.289,E2 -15571.289} C_VEL
LIN {X 0,Y 312.153,Z 527.843,A -85,B 0,C 180,E1 -15572.581,E2 -15572.581} C_VEL
LIN {X 0,Y 312.041,Z 526.487,A -85,B 0,C 180,E1 -15573.874,E2 -15573.874} C_VEL
LIN {X 0,Y 311.838,Z 523.568,A -85,B 0,C 180,E1 -15575.821,E2 -15575.821} C_VEL
LIN {X 0,Y 311.62,Z 519.499,A -85,B 0,C 180,E1 -15577.777,E2 -15577.777} C_VEL
LIN {X 0,Y 311.637,Z 513.201,A -85,B 0,C 180,E1 -15580.065,E2 -15580.065} C_VEL
LIN {X 0,Y 312.019,Z 506.323,A -85,B 0,C 180,E1 -15582.025,E2 -15582.025} C_VEL
LIN {X 0,Y 312.712,Z 497.689,A -85,B 0,C 180,E1 -15583.981,E2 -15583.981} C_VEL
LIN {X 0,Y 313.622,Z 488.903,A -85,B 0,C 180,E1 -15585.599,E2 -15585.599} C_VEL
LIN {X 0,Y 314.881,Z 478.162,A -85,B 0,C 180,E1 -15587.201,E2 -15587.201} C_VEL
LIN {X 0,Y 315.01,Z 470.162,A -85,B 0,C 180,E1 -15588.2,E2 -15588.2} C_VEL
LIN {X 0,Y 314.744,Z 458.728,A -85,B 0,C 180,E1 -15589.399,E2 -15589.399} C_VEL
LIN {X 0,Y 313.976,Z 445.504,A -85,B 0,C 180,E1 -15590.497,E2 -15590.497} C_VEL
LIN {X 0,Y 313.011,Z 432.096,A -85,B 0,C 180,E1 -15591.334,E2 -15591.334} C_VEL
LIN {X 0,Y 312.01,Z 421.404,A -85,B 0,C 180,E1 -15591.861,E2 -15591.861} C_VEL
LIN {X 0,Y 312.133,Z 419.039,A -85,B 0,C 180,E1 -15592.607,E2 -15592.607} C_VEL
LIN {X 0,Y 313.031,Z 408.185,A -85,B 0,C 180,E1 -15596.681,E2 -15596.681} C_VEL
LIN {X 0,Y 314.22,Z 396.951,A -85,B 0,C 180,E1 -15600.958,E2 -15600.958} C_VEL
LIN {X 0,Y 315.554,Z 386.81,A -85,B 0,C 180,E1 -15604.859,E2 -15604.859} C_VEL
LIN {X 0,Y 316.686,Z 379.792,A -85,B 0,C 180,E1 -15607.608,E2 -15607.608} C_VEL
LIN {X 0,Y 316.154,Z 375.243,A -85,B 0,C 180,E1 -15609.504,E2 -15609.504} C_VEL
LIN {X 0,Y 314.466,Z 366.543,A -85,B 0,C 180,E1 -15613.304,E2 -15613.304} C_VEL
LIN {X 0,Y 312.972,Z 358.995,A -85,B 0,C 180,E1 -15616.772,E2 -15616.772} C_VEL
LIN {X 0,Y 312.496,Z 356.609,A -85,B 0,C 180,E1 -15618.02,E2 -15618.02} C_VEL
LIN {X 0,Y 312.479,Z 356.56,A -85,B 0,C 180,E1 -15621.922,E2 -15621.922} C_VEL
LIN {X 0,Y 312.525,Z 356.553,A -85,B 0,C 180,E1 -15624.219,E2 -15624.219} C_VEL
LIN {X 0,Y 312.499,Z 356.561,A -85,B 0,C 180,E1 -15627.333,E2 -15627.333} C_VEL
LIN {X 0,Y 312.546,Z 356.555,A -85,B 0,C 180,E1 -15631.276,E2 -15631.276} C_VEL
LIN {X 0,Y 312.578,Z 356.548,A -85,B 0,C 180,E1 -15634.71,E2 -15634.71} C_VEL
LIN {X 0,Y 312.557,Z 356.55,A -85,B 0,C 180,E1 -15637.527,E2 -15637.527} C_VEL
LIN {X 0,Y 312.575,Z 356.547,A -85,B 0,C 180,E1 -15641.652,E2 -15641.652} C_VEL
LIN {X 0,Y 312.678,Z 356.534,A -85,B 0,C 180,E1 -15645.685,E2 -15645.685} C_VEL
LIN {X 0,Y 312.677,Z 356.534,A -85,B 0,C 180,E1 -15649.641,E2 -15649.641} C_VEL
LIN {X 0,Y 312.822,Z 356.516,A -85,B 0,C 180,E1 -15652.253,E2 -15652.253} C_VEL
LIN {X 0,Y 312.7,Z 356.536,A -85,B 0,C 180,E1 -15654.842,E2 -15654.842} C_VEL
LIN {X 0,Y 312.982,Z 356.5,A -85,B 0,C 180,E1 -15658.713,E2 -15658.713} C_VEL
LIN {X 0,Y 312.982,Z 356.497,A -85,B 0,C 180,E1 -15661.287,E2 -15661.287} C_VEL
LIN {X 0,Y 312.705,Z 356.532,A -85,B 0,C 180,E1 -15665.158,E2 -15665.158} C_VEL
LIN {X 0,Y 312.858,Z 356.511,A -85,B 0,C 180,E1 -15667.746,E2 -15667.746} C_VEL
LIN {X 0,Y 312.661,Z 356.535,A -85,B 0,C 180,E1 -15671.672,E2 -15671.672} C_VEL
LIN {X 0,Y 312.693,Z 356.534,A -85,B 0,C 180,E1 -15674.888,E2 -15674.888} C_VEL
LIN {X 0,Y 312.624,Z 356.541,A -85,B 0,C 180,E1 -15679.237,E2 -15679.237} C_VEL
LIN {X 0,Y 312.539,Z 356.553,A -85,B 0,C 180,E1 -15682.789,E2 -15682.789} C_VEL
LIN {X 0,Y 312.597,Z 356.545,A -85,B 0,C 180,E1 -15685.936,E2 -15685.936} C_VEL
LIN {X 0,Y 312.54,Z 356.551,A -85,B 0,C 180,E1 -15689.651,E2 -15689.651} C_VEL
LIN {X 0,Y 312.514,Z 356.555,A -85,B 0,C 180,E1 -15693.689,E2 -15693.689} C_VEL
LIN {X 0,Y 312.535,Z 356.551,A -85,B 0,C 180,E1 -15697.384,E2 -15697.384} C_VEL
LIN {X 0,Y 312.495,Z 356.558,A -85,B 0,C 180,E1 -15700.708,E2 -15700.708} C_VEL
LIN {X 0,Y 312.464,Z 356.565,A -85,B 0,C 180,E1 -15704.207,E2 -15704.207} C_VEL
LIN {X 0,Y 312.483,Z 356.561,A -85,B 0,C 180,E1 -15707.919,E2 -15707.919} C_VEL
LIN {X 0,Y 312.532,Z 356.556,A -85,B 0,C 180,E1 -15711.911,E2 -15711.911} C_VEL
LIN {X 0,Y 312.505,Z 356.558,A -85,B 0,C 180,E1 -15715.791,E2 -15715.791} C_VEL
LIN {X 0,Y 312.527,Z 356.552,A -85,B 0,C 180,E1 -15718.855,E2 -15718.855} C_VEL
LIN {X 0,Y 312.584,Z 356.55,A -85,B 0,C 180,E1 -15721.827,E2 -15721.827} C_VEL
LIN {X 0,Y 312.585,Z 356.545,A -85,B 0,C 180,E1 -15724.712,E2 -15724.712} C_VEL
LIN {X 0,Y 312.588,Z 356.547,A -85,B 0,C 180,E1 -15727.53,E2 -15727.53} C_VEL
LIN {X 0,Y 312.64,Z 356.542,A -85,B 0,C 180,E1 -15731.657,E2 -15731.657} C_VEL
LIN {X 0,Y 312.695,Z 356.536,A -85,B 0,C 180,E1 -15735.687,E2 -15735.687} C_VEL
LIN {X 0,Y 312.704,Z 356.535,A -85,B 0,C 180,E1 -15739.642,E2 -15739.642} C_VEL
LIN {X 0,Y 312.874,Z 356.51,A -85,B 0,C 180,E1 -15742.255,E2 -15742.255} C_VEL
LIN {X 0,Y 312.721,Z 356.528,A -85,B 0,C 180,E1 -15744.843,E2 -15744.843} C_VEL
LIN {X 0,Y 312.955,Z 356.503,A -85,B 0,C 180,E1 -15747.426,E2 -15747.426} C_VEL
LIN {X 0,Y 313.123,Z 356.48,A -85,B 0,C 180,E1 -15750,E2 -15750} C_VEL
LIN {X 0,Y 312.941,Z 356.501,A -85,B 0,C 180,E1 -15752.574,E2 -15752.574} C_VEL
LIN {X 0,Y 312.902,Z 356.505,A -85,B 0,C 180,E1 -15756.448,E2 -15756.448} C_VEL
LIN {X 0,Y 312.787,Z 356.522,A -85,B 0,C 180,E1 -15759.049,E2 -15759.049} C_VEL
LIN {X 0,Y 312.636,Z 356.541,A -85,B 0,C 180,E1 -15762.991,E2 -15762.991} C_VEL
LIN {X 0,Y 312.639,Z 356.541,A -85,B 0,C 180,E1 -15765.649,E2 -15765.649} C_VEL
LIN {X 0,Y 312.631,Z 356.545,A -85,B 0,C 180,E1 -15769.236,E2 -15769.236} C_VEL
LIN {X 0,Y 312.546,Z 356.552,A -85,B 0,C 180,E1 -15772.789,E2 -15772.789} C_VEL
LIN {X 0,Y 312.596,Z 356.544,A -85,B 0,C 180,E1 -15775.933,E2 -15775.933} C_VEL
LIN {X 0,Y 312.537,Z 356.552,A -85,B 0,C 180,E1 -15779.65,E2 -15779.65} C_VEL
LIN {X 0,Y 312.518,Z 356.554,A -85,B 0,C 180,E1 -15783.688,E2 -15783.688} C_VEL
LIN {X 0,Y 312.551,Z 356.552,A -85,B 0,C 180,E1 -15787.38,E2 -15787.38} C_VEL
LIN {X 0,Y 312.582,Z 356.687,A -85,B 0,C 180,E1 -15791.495,E2 -15791.495} C_VEL
LIN {X 0,Y 312.876,Z 357.853,A -85,B 0,C 180,E1 -15791.742,E2 -15791.742} C_VEL
LIN {X 0,Y 316.536,Z 370.509,A -85,B 0,C 180,E1 -15793.031,E2 -15793.031} C_VEL
LIN {X 0,Y 318.668,Z 378.683,A -85,B 0,C 180,E1 -15794.003,E2 -15794.003} C_VEL
LIN {X 0,Y 317.72,Z 390.027,A -85,B 0,C 180,E1 -15795.395,E2 -15795.395} C_VEL
LIN {X 0,Y 316.716,Z 399.96,A -85,B 0,C 180,E1 -15796.891,E2 -15796.891} C_VEL
LIN {X 0,Y 315.801,Z 408.496,A -85,B 0,C 180,E1 -15798.45,E2 -15798.45} C_VEL
LIN {X 0,Y 315.002,Z 415.985,A -85,B 0,C 180,E1 -15800.101,E2 -15800.101} C_VEL
LIN {X 0,Y 314.233,Z 423.469,A -85,B 0,C 180,E1 -15802.139,E2 -15802.139} C_VEL
LIN {X 0,Y 313.513,Z 429.907,A -85,B 0,C 180,E1 -15804.349,E2 -15804.349} C_VEL
LIN {X 0,Y 313.07,Z 435.124,A -85,B 0,C 180,E1 -15806.758,E2 -15806.758} C_VEL
LIN {X 0,Y 312.833,Z 438.418,A -85,B 0,C 180,E1 -15808.888,E2 -15808.888} C_VEL
LIN {X 0,Y 312.798,Z 440.695,A -85,B 0,C 180,E1 -15811.192,E2 -15811.192} C_VEL
LIN {X 0,Y 313.028,Z 441.692,A -85,B 0,C 180,E1 -15813.902,E2 -15813.902} C_VEL
LIN {X 0,Y 313.521,Z 441.184,A -85,B 0,C 180,E1 -15816.203,E2 -15816.203} C_VEL
LIN {X 0,Y 313.959,Z 440.204,A -85,B 0,C 180,E1 -15817.632,E2 -15817.632} C_VEL
LIN {X 0,Y 314.777,Z 437.922,A -85,B 0,C 180,E1 -15819.67,E2 -15819.67} C_VEL
LIN {X 0,Y 315.76,Z 434.287,A -85,B 0,C 180,E1 -15821.844,E2 -15821.844} C_VEL
LIN {X 0,Y 317.038,Z 429.505,A -85,B 0,C 180,E1 -15823.913,E2 -15823.913} C_VEL
LIN {X 0,Y 318.551,Z 423.345,A -85,B 0,C 180,E1 -15825.955,E2 -15825.955} C_VEL
LIN {X 0,Y 320.255,Z 415.698,A -85,B 0,C 180,E1 -15827.936,E2 -15827.936} C_VEL
LIN {X 0,Y 320.389,Z 412.204,A -85,B 0,C 180,E1 -15828.791,E2 -15828.791} C_VEL
LIN {X 0,Y 319.119,Z 406.456,A -85,B 0,C 180,E1 -15830.222,E2 -15830.222} C_VEL
LIN {X 0,Y 317.842,Z 400.154,A -85,B 0,C 180,E1 -15831.573,E2 -15831.573} C_VEL
LIN {X 0,Y 317.938,Z 395.799,A -85,B 0,C 180,E1 -15832.289,E2 -15832.289} C_VEL
LIN {X 0,Y 318.623,Z 391.543,A -85,B 0,C 180,E1 -15832.873,E2 -15832.873} C_VEL
LIN {X 0,Y 316.55,Z 382.826,A -85,B 0,C 180,E1 -15834.34,E2 -15834.34} C_VEL
LIN {X 0,Y 313.326,Z 373.759,A -85,B 0,C 180,E1 -15835.82,E2 -15835.82} C_VEL
LIN {X 0,Y 308.286,Z 362.914,A -85,B 0,C 180,E1 -15837.55,E2 -15837.55} C_VEL
LIN {X 0,Y 306.061,Z 358.119,A -85,B 0,C 180,E1 -15838.314,E2 -15838.314} C_VEL
LIN {X 0,Y 305.949,Z 357.402,A -85,B 0,C 180,E1 -15838.684,E2 -15838.684} C_VEL
LIN {X 0,Y 305.949,Z 357.369,A -85,B 0,C 180,E1 -15841.316,E2 -15841.316} C_VEL
LIN {X 0,Y 305.673,Z 357.409,A -85,B 0,C 180,E1 -15845.277,E2 -15845.277} C_VEL
LIN {X 0,Y 305.763,Z 357.397,A -85,B 0,C 180,E1 -15847.927,E2 -15847.927} C_VEL
LIN {X 0,Y 305.591,Z 357.417,A -85,B 0,C 180,E1 -15851.946,E2 -15851.946} C_VEL
LIN {X 0,Y 305.601,Z 357.419,A -85,B 0,C 180,E1 -15855.014,E2 -15855.014} C_VEL
LIN {X 0,Y 305.536,Z 357.427,A -85,B 0,C 180,E1 -15859.427,E2 -15859.427} C_VEL
LIN {X 0,Y 305.48,Z 357.429,A -85,B 0,C 180,E1 -15863.04,E2 -15863.04} C_VEL
LIN {X 0,Y 305.519,Z 357.423,A -85,B 0,C 180,E1 -15866.219,E2 -15866.219} C_VEL
LIN {X 0,Y 305.482,Z 357.429,A -85,B 0,C 180,E1 -15869.048,E2 -15869.048} C_VEL
LIN {X 0,Y 305.437,Z 357.438,A -85,B 0,C 180,E1 -15871.953,E2 -15871.953} C_VEL
LIN {X 0,Y 305.504,Z 357.506,A -85,B 0,C 180,E1 -15875.921,E2 -15875.921} C_VEL
LIN {X 0,Y 306.493,Z 362.347,A -85,B 0,C 180,E1 -15879.945,E2 -15879.945} C_VEL
LIN {X 0,Y 307.528,Z 367.105,A -85,B 0,C 180,E1 -15883.283,E2 -15883.283} C_VEL
LIN {X 0,Y 308.661,Z 372.771,A -85,B 0,C 180,E1 -15886.771,E2 -15886.771} C_VEL
LIN {X 0,Y 309.643,Z 378.097,A -85,B 0,C 180,E1 -15889.696,E2 -15889.696} C_VEL
LIN {X 0,Y 310.113,Z 381.541,A -85,B 0,C 180,E1 -15891.449,E2 -15891.449} C_VEL
LIN {X 0,Y 309.52,Z 385.354,A -85,B 0,C 180,E1 -15893.164,E2 -15893.164} C_VEL
LIN {X 0,Y 307.84,Z 395.034,A -85,B 0,C 180,E1 -15897.311,E2 -15897.311} C_VEL
LIN {X 0,Y 306.535,Z 404.665,A -85,B 0,C 180,E1 -15901.219,E2 -15901.219} C_VEL
LIN {X 0,Y 306.069,Z 409.463,A -85,B 0,C 180,E1 -15903.004,E2 -15903.004} C_VEL
LIN {X 0,Y 307.905,Z 417.585,A -85,B 0,C 180,E1 -15903.708,E2 -15903.708} C_VEL
LIN {X 0,Y 310.454,Z 431.385,A -85,B 0,C 180,E1 -15904.893,E2 -15904.893} C_VEL
LIN {X 0,Y 311.75,Z 443.718,A -85,B 0,C 180,E1 -15906.06,E2 -15906.06} C_VEL
LIN {X 0,Y 311.969,Z 456.969,A -85,B 0,C 180,E1 -15907.465,E2 -15907.465} C_VEL
LIN {X 0,Y 311.15,Z 469.407,A -85,B 0,C 180,E1 -15908.988,E2 -15908.988} C_VEL
LIN {X 0,Y 310.241,Z 479.564,A -85,B 0,C 180,E1 -15910.48,E2 -15910.48} C_VEL
LIN {X 0,Y 308.457,Z 488.973,A -85,B 0,C 180,E1 -15912.086,E2 -15912.086} C_VEL
LIN {X 0,Y 306.756,Z 498.336,A -85,B 0,C 180,E1 -15914.043,E2 -15914.043} C_VEL
LIN {X 0,Y 305.612,Z 506.099,A -85,B 0,C 180,E1 -15916.027,E2 -15916.027} C_VEL
LIN {X 0,Y 304.778,Z 512.465,A -85,B 0,C 180,E1 -15918.022,E2 -15918.022} C_VEL
LIN {X 0,Y 304.326,Z 517.617,A -85,B 0,C 180,E1 -15920.026,E2 -15920.026} C_VEL
LIN {X 0,Y 304.273,Z 521.683,A -85,B 0,C 180,E1 -15922.034,E2 -15922.034} C_VEL
LIN {X 0,Y 304.431,Z 523.84,A -85,B 0,C 180,E1 -15923.372,E2 -15923.372} C_VEL
LIN {X 0,Y 304.893,Z 526.851,A -85,B 0,C 180,E1 -15926.035,E2 -15926.035} C_VEL
LIN {X 0,Y 304.995,Z 527.714,A -85,B 0,C 180,E1 -15927.359,E2 -15927.359} C_VEL
LIN {X 0,Y 305.404,Z 528.155,A -85,B 0,C 180,E1 -15928.681,E2 -15928.681} C_VEL
LIN {X 0,Y 305.681,Z 528.148,A -85,B 0,C 180,E1 -15930,E2 -15930} C_VEL
LIN {X 0,Y 305.433,Z 527.644,A -85,B 0,C 180,E1 -15931.318,E2 -15931.318} C_VEL
LIN {X 0,Y 305.117,Z 526.697,A -85,B 0,C 180,E1 -15932.64,E2 -15932.64} C_VEL
LIN {X 0,Y 304.995,Z 525.284,A -85,B 0,C 180,E1 -15933.964,E2 -15933.964} C_VEL
LIN {X 0,Y 304.784,Z 522.298,A -85,B 0,C 180,E1 -15935.956,E2 -15935.956} C_VEL
LIN {X 0,Y 304.543,Z 518.151,A -85,B 0,C 180,E1 -15937.959,E2 -15937.959} C_VEL
LIN {X 0,Y 304.61,Z 511.781,A -85,B 0,C 180,E1 -15940.3,E2 -15940.3} C_VEL
LIN {X 0,Y 304.985,Z 504.765,A -85,B 0,C 180,E1 -15942.307,E2 -15942.307} C_VEL
LIN {X 0,Y 305.758,Z 496.022,A -85,B 0,C 180,E1 -15944.305,E2 -15944.305} C_VEL
LIN {X 0,Y 306.86,Z 486.137,A -85,B 0,C 180,E1 -15946.122,E2 -15946.122} C_VEL
LIN {X 0,Y 308.059,Z 474.871,A -85,B 0,C 180,E1 -15947.766,E2 -15947.766} C_VEL
LIN {X 0,Y 307.86,Z 463.2,A -85,B 0,C 180,E1 -15949.157,E2 -15949.157} C_VEL
LIN {X 0,Y 307.278,Z 450.915,A -85,B 0,C 180,E1 -15950.323,E2 -15950.323} C_VEL
LIN {X 0,Y 306.526,Z 438.313,A -85,B 0,C 180,E1 -15951.262,E2 -15951.262} C_VEL
LIN {X 0,Y 305.343,Z 424.666,A -85,B 0,C 180,E1 -15952.015,E2 -15952.015} C_VEL
LIN {X 0,Y 304.981,Z 420.402,A -85,B 0,C 180,E1 -15952.244,E2 -15952.244} C_VEL
LIN {X 0,Y 305.268,Z 416.17,A -85,B 0,C 180,E1 -15953.758,E2 -15953.758} C_VEL
LIN {X 0,Y 306.301,Z 405.055,A -85,B 0,C 180,E1 -15958.057,E2 -15958.057} C_VEL
LIN {X 0,Y 307.72,Z 393.201,A -85,B 0,C 180,E1 -15962.697,E2 -15962.697} C_VEL
LIN {X 0,Y 309.544,Z 381.461,A -85,B 0,C 180,E1 -15967.377,E2 -15967.377} C_VEL
LIN {X 0,Y 309.535,Z 378.59,A -85,B 0,C 180,E1 -15968.574,E2 -15968.574} C_VEL
LIN {X 0,Y 308.324,Z 372.197,A -85,B 0,C 180,E1 -15971.377,E2 -15971.377} C_VEL
LIN {X 0,Y 306.698,Z 363.699,A -85,B 0,C 180,E1 -15975.263,E2 -15975.263} C_VEL
LIN {X 0,Y 305.455,Z 357.503,A -85,B 0,C 180,E1 -15978.32,E2 -15978.32} C_VEL
LIN {X 0,Y 305.455,Z 357.437,A -85,B 0,C 180,E1 -15981.594,E2 -15981.594} C_VEL
LIN {X 0,Y 305.456,Z 357.435,A -85,B 0,C 180,E1 -15984.886,E2 -15984.886} C_VEL
LIN {X 0,Y 305.446,Z 357.434,A -85,B 0,C 180,E1 -15988.354,E2 -15988.354} C_VEL
LIN {X 0,Y 305.515,Z 357.43,A -85,B 0,C 180,E1 -15991.113,E2 -15991.113} C_VEL
LIN {X 0,Y 305.559,Z 357.42,A -85,B 0,C 180,E1 -15994.087,E2 -15994.087} C_VEL
LIN {X 0,Y 305.468,Z 357.431,A -85,B 0,C 180,E1 -15998.4,E2 -15998.4} C_VEL
LIN {X 0,Y 305.536,Z 357.427,A -85,B 0,C 180,E1 -16001.214,E2 -16001.214} C_VEL
LIN {X 0,Y 305.619,Z 357.414,A -85,B 0,C 180,E1 -16005.347,E2 -16005.347} C_VEL
LIN {X 0,Y 305.616,Z 357.415,A -85,B 0,C 180,E1 -16009.399,E2 -16009.399} C_VEL
LIN {X 0,Y 305.763,Z 357.395,A -85,B 0,C 180,E1 -16012.073,E2 -16012.073} C_VEL
LIN {X 0,Y 305.67,Z 357.41,A -85,B 0,C 180,E1 -16014.723,E2 -16014.723} C_VEL
LIN {X 0,Y 305.949,Z 357.376,A -85,B 0,C 180,E1 -16018.684,E2 -16018.684} C_VEL
LIN {X 0,Y 305.948,Z 357.373,A -85,B 0,C 180,E1 -16021.316,E2 -16021.316} C_VEL
LIN {X 0,Y 305.838,Z 357.389,A -85,B 0,C 180,E1 -16026.598,E2 -16026.598} C_VEL
LIN {X 0,Y 305.729,Z 357.4,A -85,B 0,C 180,E1 -16029.26,E2 -16029.26} C_VEL
LIN {X 0,Y 305.581,Z 357.418,A -85,B 0,C 180,E1 -16033.296,E2 -16033.296} C_VEL
LIN {X 0,Y 305.587,Z 357.418,A -85,B 0,C 180,E1 -16036.02,E2 -16036.02} C_VEL
LIN {X 0,Y 305.57,Z 357.419,A -85,B 0,C 180,E1 -16039.445,E2 -16039.445} C_VEL
LIN {X 0,Y 305.484,Z 357.431,A -85,B 0,C 180,E1 -16043.042,E2 -16043.042} C_VEL
LIN {X 0,Y 305.542,Z 357.426,A -85,B 0,C 180,E1 -16046.228,E2 -16046.228} C_VEL
LIN {X 0,Y 305.49,Z 357.429,A -85,B 0,C 180,E1 -16049.05,E2 -16049.05} C_VEL
LIN {X 0,Y 305.46,Z 357.433,A -85,B 0,C 180,E1 -16053.518,E2 -16053.518} C_VEL
LIN {X 0,Y 305.492,Z 357.43,A -85,B 0,C 180,E1 -16056.737,E2 -16056.737} C_VEL
LIN {X 0,Y 305.458,Z 357.435,A -85,B 0,C 180,E1 -16060.602,E2 -16060.602} C_VEL
LIN {X 0,Y 305.443,Z 357.436,A -85,B 0,C 180,E1 -16063.652,E2 -16063.652} C_VEL
LIN {X 0,Y 305.455,Z 357.433,A -85,B 0,C 180,E1 -16067.414,E2 -16067.414} C_VEL
LIN {X 0,Y 305.493,Z 357.43,A -85,B 0,C 180,E1 -16071.601,E2 -16071.601} C_VEL
LIN {X 0,Y 305.461,Z 357.432,A -85,B 0,C 180,E1 -16074.888,E2 -16074.888} C_VEL
LIN {X 0,Y 305.455,Z 357.435,A -85,B 0,C 180,E1 -16078.354,E2 -16078.354} C_VEL
LIN {X 0,Y 305.528,Z 357.424,A -85,B 0,C 180,E1 -16081.115,E2 -16081.115} C_VEL
LIN {X 0,Y 305.572,Z 357.422,A -85,B 0,C 180,E1 -16084.089,E2 -16084.089} C_VEL
LIN {X 0,Y 305.501,Z 357.428,A -85,B 0,C 180,E1 -16088.403,E2 -16088.403} C_VEL
LIN {X 0,Y 305.591,Z 357.417,A -85,B 0,C 180,E1 -16091.218,E2 -16091.218} C_VEL
LIN {X 0,Y 305.65,Z 357.411,A -85,B 0,C 180,E1 -16095.349,E2 -16095.349} C_VEL
LIN {X 0,Y 305.64,Z 357.413,A -85,B 0,C 180,E1 -16099.4,E2 -16099.4} C_VEL
LIN {X 0,Y 305.815,Z 357.39,A -85,B 0,C 180,E1 -16102.075,E2 -16102.075} C_VEL
LIN {X 0,Y 305.692,Z 357.404,A -85,B 0,C 180,E1 -16104.724,E2 -16104.724} C_VEL
LIN {X 0,Y 305.962,Z 357.37,A -85,B 0,C 180,E1 -16108.684,E2 -16108.684} C_VEL
LIN {X 0,Y 305.96,Z 357.374,A -85,B 0,C 180,E1 -16111.316,E2 -16111.316} C_VEL
LIN {X 0,Y 305.689,Z 357.407,A -85,B 0,C 180,E1 -16115.276,E2 -16115.276} C_VEL
LIN {X 0,Y 305.798,Z 357.392,A -85,B 0,C 180,E1 -16117.926,E2 -16117.926} C_VEL
LIN {X 0,Y 305.605,Z 357.415,A -85,B 0,C 180,E1 -16121.945,E2 -16121.945} C_VEL
LIN {X 0,Y 305.639,Z 357.413,A -85,B 0,C 180,E1 -16125.035,E2 -16125.035} C_VEL
LIN {X 0,Y 305.577,Z 357.422,A -85,B 0,C 180,E1 -16129.445,E2 -16129.445} C_VEL
LIN {X 0,Y 305.491,Z 357.433,A -85,B 0,C 180,E1 -16133.041,E2 -16133.041} C_VEL
LIN {X 0,Y 305.525,Z 357.424,A -85,B 0,C 180,E1 -16136.218,E2 -16136.218} C_VEL
LIN {X 0,Y 305.488,Z 357.434,A -85,B 0,C 180,E1 -16139.047,E2 -16139.047} C_VEL
LIN {X 0,Y 305.441,Z 357.436,A -85,B 0,C 180,E1 -16141.952,E2 -16141.952} C_VEL
LIN {X 0,Y 305.461,Z 357.438,A -85,B 0,C 180,E1 -16145.112,E2 -16145.112} C_VEL
LIN {X 0,Y 305.492,Z 357.431,A -85,B 0,C 180,E1 -16148.539,E2 -16148.539} C_VEL
LIN {X 0,Y 305.565,Z 357.653,A -85,B 0,C 180,E1 -16151.186,E2 -16151.186} C_VEL
LIN {X 0,Y 305.851,Z 358.831,A -85,B 0,C 180,E1 -16151.416,E2 -16151.416} C_VEL
LIN {X 0,Y 309.217,Z 370.39,A -85,B 0,C 180,E1 -16152.596,E2 -16152.596} C_VEL
LIN {X 0,Y 311.712,Z 380.486,A -85,B 0,C 180,E1 -16153.823,E2 -16153.823} C_VEL
LIN {X 0,Y 310.721,Z 391.856,A -85,B 0,C 180,E1 -16155.271,E2 -16155.271} C_VEL
LIN {X 0,Y 309.691,Z 401.635,A -85,B 0,C 180,E1 -16156.795,E2 -16156.795} C_VEL
LIN {X 0,Y 308.63,Z 411.358,A -85,B 0,C 180,E1 -16158.671,E2 -16158.671} C_VEL
LIN {X 0,Y 307.692,Z 419.741,A -85,B 0,C 180,E1 -16160.676,E2 -16160.676} C_VEL
LIN {X 0,Y 306.983,Z 426.356,A -85,B 0,C 180,E1 -16162.644,E2 -16162.644} C_VEL
LIN {X 0,Y 306.319,Z 432.537,A -85,B 0,C 180,E1 -16164.999,E2 -16164.999} C_VEL
LIN {X 0,Y 305.982,Z 437.125,A -85,B 0,C 180,E1 -16167.332,E2 -16167.332} C_VEL
LIN {X 0,Y 305.757,Z 440.237,A -85,B 0,C 180,E1 -16169.623,E2 -16169.623} C_VEL
LIN {X 0,Y 305.773,Z 441.608,A -85,B 0,C 180,E1 -16171.14,E2 -16171.14} C_VEL
LIN {X 0,Y 305.956,Z 442.733,A -85,B 0,C 180,E1 -16173.615,E2 -16173.615} C_VEL
LIN {X 0,Y 306.353,Z 442.602,A -85,B 0,C 180,E1 -16175.611,E2 -16175.611} C_VEL
LIN {X 0,Y 306.759,Z 441.891,A -85,B 0,C 180,E1 -16177.078,E2 -16177.078} C_VEL
LIN {X 0,Y 307.702,Z 439.694,A -85,B 0,C 180,E1 -16179.46,E2 -16179.46} C_VEL
LIN {X 0,Y 308.576,Z 436.87,A -85,B 0,C 180,E1 -16181.406,E2 -16181.406} C_VEL
LIN {X 0,Y 309.83,Z 432.614,A -85,B 0,C 180,E1 -16183.528,E2 -16183.528} C_VEL
LIN {X 0,Y 311.347,Z 426.986,A -85,B 0,C 180,E1 -16185.623,E2 -16185.623} C_VEL
LIN {X 0,Y 313.089,Z 419.87,A -85,B 0,C 180,E1 -16187.687,E2 -16187.687} C_VEL
LIN {X 0,Y 314.677,Z 412.855,A -85,B 0,C 180,E1 -16189.318,E2 -16189.318} C_VEL
LIN {X 0,Y 316.549,Z 403.656,A -85,B 0,C 180,E1 -16191.059,E2 -16191.059} C_VEL
LIN {X 0,Y 317.938,Z 395.799,A -85,B 0,C 180,E1 -16192.289,E2 -16192.289} C_VEL
LIN {X 0,Y 317.898,Z 392.911,A -85,B 0,C 180,E1 -16192.755,E2 -16192.755} C_VEL
LIN {X 0,Y 316.537,Z 389.014,A -85,B 0,C 180,E1 -16193.521,E2 -16193.521} C_VEL
LIN {X 0,Y 314.22,Z 385.647,A -85,B 0,C 180,E1 -16194.312,E2 -16194.312} C_VEL
LIN {X 0,Y 308.645,Z 378.888,A -85,B 0,C 180,E1 -16195.93,E2 -16195.93} C_VEL
LIN {X 0,Y 307.115,Z 376.232,A -85,B 0,C 180,E1 -16196.443,E2 -16196.443} C_VEL
LIN {X 0,Y 301.681,Z 364.335,A -85,B 0,C 180,E1 -16198.454,E2 -16198.454} C_VEL
LIN {X 0,Y 299.064,Z 358.923,A -85,B 0,C 180,E1 -16199.369,E2 -16199.369} C_VEL
LIN {X 0,Y 298.987,Z 358.251,A -85,B 0,C 180,E1 -16199.832,E2 -16199.832} C_VEL
LIN {X 0,Y 298.826,Z 358.264,A -85,B 0,C 180,E1 -16202.696,E2 -16202.696} C_VEL
LIN {X 0,Y 298.767,Z 358.269,A -85,B 0,C 180,E1 -16206.755,E2 -16206.755} C_VEL
LIN {X 0,Y 298.618,Z 358.288,A -85,B 0,C 180,E1 -16209.483,E2 -16209.483} C_VEL
LIN {X 0,Y 298.538,Z 358.297,A -85,B 0,C 180,E1 -16213.616,E2 -16213.616} C_VEL
LIN {X 0,Y 298.479,Z 358.306,A -85,B 0,C 180,E1 -16216.413,E2 -16216.413} C_VEL
LIN {X 0,Y 298.476,Z 358.305,A -85,B 0,C 180,E1 -16219.639,E2 -16219.639} C_VEL
LIN {X 0,Y 298.423,Z 358.306,A -85,B 0,C 180,E1 -16223.601,E2 -16223.601} C_VEL
LIN {X 0,Y 298.48,Z 358.3,A -85,B 0,C 180,E1 -16226.575,E2 -16226.575} C_VEL
LIN {X 0,Y 298.411,Z 358.313,A -85,B 0,C 180,E1 -16229.642,E2 -16229.642} C_VEL
LIN {X 0,Y 298.39,Z 358.315,A -85,B 0,C 180,E1 -16232.801,E2 -16232.801} C_VEL
LIN {X 0,Y 298.425,Z 358.388,A -85,B 0,C 180,E1 -16234.601,E2 -16234.601} C_VEL
LIN {X 0,Y 299.117,Z 361.68,A -85,B 0,C 180,E1 -16237.654,E2 -16237.654} C_VEL
LIN {X 0,Y 300.197,Z 366.569,A -85,B 0,C 180,E1 -16241.484,E2 -16241.484} C_VEL
LIN {X 0,Y 301.105,Z 370.912,A -85,B 0,C 180,E1 -16244.445,E2 -16244.445} C_VEL
LIN {X 0,Y 302.264,Z 376.953,A -85,B 0,C 180,E1 -16248.077,E2 -16248.077} C_VEL
LIN {X 0,Y 303.084,Z 381.647,A -85,B 0,C 180,E1 -16250.624,E2 -16250.624} C_VEL
LIN {X 0,Y 303.079,Z 384.49,A -85,B 0,C 180,E1 -16252.038,E2 -16252.038} C_VEL
LIN {X 0,Y 301.064,Z 394.972,A -85,B 0,C 180,E1 -16256.681,E2 -16256.681} C_VEL
LIN {X 0,Y 299.486,Z 405.879,A -85,B 0,C 180,E1 -16261.245,E2 -16261.245} C_VEL
LIN {X 0,Y 299.268,Z 408.034,A -85,B 0,C 180,E1 -16261.987,E2 -16261.987} C_VEL
LIN {X 0,Y 300.618,Z 413.897,A -85,B 0,C 180,E1 -16262.546,E2 -16262.546} C_VEL
LIN {X 0,Y 303.275,Z 426.473,A -85,B 0,C 180,E1 -16263.693,E2 -16263.693} C_VEL
LIN {X 0,Y 305.139,Z 441.546,A -85,B 0,C 180,E1 -16265.177,E2 -16265.177} C_VEL
LIN {X 0,Y 305.521,Z 453.239,A -85,B 0,C 180,E1 -16266.442,E2 -16266.442} C_VEL
LIN {X 0,Y 304.95,Z 464.65,A -85,B 0,C 180,E1 -16267.834,E2 -16267.834} C_VEL
LIN {X 0,Y 303.655,Z 477.394,A -85,B 0,C 180,E1 -16269.686,E2 -16269.686} C_VEL
LIN {X 0,Y 302.451,Z 485.189,A -85,B 0,C 180,E1 -16271.016,E2 -16271.016} C_VEL
LIN {X 0,Y 300.739,Z 493.523,A -85,B 0,C 180,E1 -16272.666,E2 -16272.666} C_VEL
LIN {X 0,Y 299.237,Z 501.293,A -85,B 0,C 180,E1 -16274.52,E2 -16274.52} C_VEL
LIN {X 0,Y 298.457,Z 506.614,A -85,B 0,C 180,E1 -16276.033,E2 -16276.033} C_VEL
LIN {X 0,Y 297.557,Z 513.563,A -85,B 0,C 180,E1 -16278.419,E2 -16278.419} C_VEL
LIN {X 0,Y 297.206,Z 518.268,A -85,B 0,C 180,E1 -16280.472,E2 -16280.472} C_VEL
LIN {X 0,Y 297.193,Z 520.84,A -85,B 0,C 180,E1 -16281.843,E2 -16281.843} C_VEL
LIN {X 0,Y 297.349,Z 522.934,A -85,B 0,C 180,E1 -16283.213,E2 -16283.213} C_VEL
LIN {X 0,Y 297.817,Z 525.884,A -85,B 0,C 180,E1 -16285.94,E2 -16285.94} C_VEL
LIN {X 0,Y 297.948,Z 526.702,A -85,B 0,C 180,E1 -16287.296,E2 -16287.296} C_VEL
LIN {X 0,Y 298.367,Z 527.104,A -85,B 0,C 180,E1 -16288.65,E2 -16288.65} C_VEL
LIN {X 0,Y 298.66,Z 527.073,A -85,B 0,C 180,E1 -16290,E2 -16290} C_VEL
LIN {X 0,Y 298.402,Z 526.54,A -85,B 0,C 180,E1 -16291.35,E2 -16291.35} C_VEL
LIN {X 0,Y 298.083,Z 525.527,A -85,B 0,C 180,E1 -16292.703,E2 -16292.703} C_VEL
LIN {X 0,Y 297.949,Z 524.074,A -85,B 0,C 180,E1 -16294.058,E2 -16294.058} C_VEL
LIN {X 0,Y 297.709,Z 521.01,A -85,B 0,C 180,E1 -16296.098,E2 -16296.098} C_VEL
LIN {X 0,Y 297.503,Z 516.789,A -85,B 0,C 180,E1 -16298.148,E2 -16298.148} C_VEL
LIN {X 0,Y 297.556,Z 511.337,A -85,B 0,C 180,E1 -16300.203,E2 -16300.203} C_VEL
LIN {X 0,Y 297.891,Z 504.489,A -85,B 0,C 180,E1 -16302.259,E2 -16302.259} C_VEL
LIN {X 0,Y 298.499,Z 497.503,A -85,B 0,C 180,E1 -16303.965,E2 -16303.965} C_VEL
LIN {X 0,Y 299.541,Z 488.006,A -85,B 0,C 180,E1 -16305.852,E2 -16305.852} C_VEL
LIN {X 0,Y 300.794,Z 477.7,A -85,B 0,C 180,E1 -16307.507,E2 -16307.507} C_VEL
LIN {X 0,Y 300.907,Z 467.056,A -85,B 0,C 180,E1 -16308.908,E2 -16308.908} C_VEL
LIN {X 0,Y 300.445,Z 455.157,A -85,B 0,C 180,E1 -16310.183,E2 -16310.183} C_VEL
LIN {X 0,Y 299.763,Z 441.894,A -85,B 0,C 180,E1 -16311.308,E2 -16311.308} C_VEL
LIN {X 0,Y 298.746,Z 428.665,A -85,B 0,C 180,E1 -16312.145,E2 -16312.145} C_VEL
LIN {X 0,Y 297.974,Z 419.551,A -85,B 0,C 180,E1 -16312.629,E2 -16312.629} C_VEL
LIN {X 0,Y 298.155,Z 416.693,A -85,B 0,C 180,E1 -16313.622,E2 -16313.622} C_VEL
LIN {X 0,Y 299.189,Z 405.592,A -85,B 0,C 180,E1 -16318.021,E2 -16318.021} C_VEL
LIN {X 0,Y 300.661,Z 393.98,A -85,B 0,C 180,E1 -16322.7,E2 -16322.7} C_VEL
LIN {X 0,Y 302.364,Z 382.992,A -85,B 0,C 180,E1 -16327.18,E2 -16327.18} C_VEL
LIN {X 0,Y 302.559,Z 380.366,A -85,B 0,C 180,E1 -16328.29,E2 -16328.29} C_VEL
LIN {X 0,Y 301.636,Z 374.896,A -85,B 0,C 180,E1 -16330.721,E2 -16330.721} C_VEL
LIN {X 0,Y 300.009,Z 366.441,A -85,B 0,C 180,E1 -16334.649,E2 -16334.649} C_VEL
LIN {X 0,Y 298.393,Z 358.396,A -85,B 0,C 180,E1 -16338.627,E2 -16338.627} C_VEL
LIN {X 0,Y 298.398,Z 358.313,A -85,B 0,C 180,E1 -16342.239,E2 -16342.239} C_VEL
LIN {X 0,Y 298.403,Z 358.315,A -85,B 0,C 180,E1 -16345.58,E2 -16345.58} C_VEL
LIN {X 0,Y 298.39,Z 358.315,A -85,B 0,C 180,E1 -16348.79,E2 -16348.79} C_VEL
LIN {X 0,Y 298.456,Z 358.305,A -85,B 0,C 180,E1 -16351.903,E2 -16351.903} C_VEL
LIN {X 0,Y 298.475,Z 358.306,A -85,B 0,C 180,E1 -16354.923,E2 -16354.923} C_VEL
LIN {X 0,Y 298.423,Z 358.313,A -85,B 0,C 180,E1 -16359.313,E2 -16359.313} C_VEL
LIN {X 0,Y 298.471,Z 358.303,A -85,B 0,C 180,E1 -16362.175,E2 -16362.175} C_VEL
LIN {X 0,Y 298.579,Z 358.294,A -85,B 0,C 180,E1 -16364.994,E2 -16364.994} C_VEL
LIN {X 0,Y 298.575,Z 358.293,A -85,B 0,C 180,E1 -16369.146,E2 -16369.146} C_VEL
LIN {X 0,Y 298.709,Z 358.274,A -85,B 0,C 180,E1 -16371.885,E2 -16371.885} C_VEL
LIN {X 0,Y 298.64,Z 358.285,A -85,B 0,C 180,E1 -16374.598,E2 -16374.598} C_VEL
LIN {X 0,Y 298.915,Z 358.251,A -85,B 0,C 180,E1 -16378.653,E2 -16378.653} C_VEL
LIN {X 0,Y 298.915,Z 358.249,A -85,B 0,C 180,E1 -16381.347,E2 -16381.347} C_VEL
LIN {X 0,Y 298.784,Z 358.269,A -85,B 0,C 180,E1 -16386.754,E2 -16386.754} C_VEL
LIN {X 0,Y 298.674,Z 358.278,A -85,B 0,C 180,E1 -16389.481,E2 -16389.481} C_VEL
LIN {X 0,Y 298.545,Z 358.293,A -85,B 0,C 180,E1 -16393.616,E2 -16393.616} C_VEL
LIN {X 0,Y 298.542,Z 358.298,A -85,B 0,C 180,E1 -16396.409,E2 -16396.409} C_VEL
LIN {X 0,Y 298.505,Z 358.299,A -85,B 0,C 180,E1 -16399.655,E2 -16399.655} C_VEL
LIN {X 0,Y 298.451,Z 358.306,A -85,B 0,C 180,E1 -16403.598,E2 -16403.598} C_VEL
LIN {X 0,Y 298.484,Z 358.306,A -85,B 0,C 180,E1 -16406.575,E2 -16406.575} C_VEL
LIN {X 0,Y 298.416,Z 358.31,A -85,B 0,C 180,E1 -16409.642,E2 -16409.642} C_VEL
LIN {X 0,Y 298.39,Z 358.315,A -85,B 0,C 180,E1 -16412.801,E2 -16412.801} C_VEL
LIN {X 0,Y 298.461,Z 358.305,A -85,B 0,C 180,E1 -16416.813,E2 -16416.813} C_VEL
LIN {X 0,Y 298.413,Z 358.311,A -85,B 0,C 180,E1 -16421.095,E2 -16421.095} C_VEL
LIN {X 0,Y 298.422,Z 358.309,A -85,B 0,C 180,E1 -16423.11,E2 -16423.11} C_VEL
LIN {X 0,Y 298.4,Z 358.312,A -85,B 0,C 180,E1 -16426.922,E2 -16426.922} C_VEL
LIN {X 0,Y 298.413,Z 358.311,A -85,B 0,C 180,E1 -16431.004,E2 -16431.004} C_VEL
LIN {X 0,Y 298.419,Z 358.314,A -85,B 0,C 180,E1 -16433.931,E2 -16433.931} C_VEL
LIN {X 0,Y 298.398,Z 358.318,A -85,B 0,C 180,E1 -16437.983,E2 -16437.983} C_VEL
LIN {X 0,Y 298.47,Z 358.308,A -85,B 0,C 180,E1 -16441.906,E2 -16441.906} C_VEL
LIN {X 0,Y 298.486,Z 358.301,A -85,B 0,C 180,E1 -16444.925,E2 -16444.925} C_VEL
LIN {X 0,Y 298.451,Z 358.307,A -85,B 0,C 180,E1 -16449.316,E2 -16449.316} C_VEL
LIN {X 0,Y 298.539,Z 358.297,A -85,B 0,C 180,E1 -16452.18,E2 -16452.18} C_VEL
LIN {X 0,Y 298.595,Z 358.288,A -85,B 0,C 180,E1 -16454.995,E2 -16454.995} C_VEL
LIN {X 0,Y 298.595,Z 358.288,A -85,B 0,C 180,E1 -16459.147,E2 -16459.147} C_VEL
LIN {X 0,Y 298.761,Z 358.27,A -85,B 0,C 180,E1 -16461.886,E2 -16461.886} C_VEL
LIN {X 0,Y 298.663,Z 358.279,A -85,B 0,C 180,E1 -16464.599,E2 -16464.599} C_VEL
LIN {X 0,Y 298.928,Z 358.246,A -85,B 0,C 180,E1 -16468.653,E2 -16468.653} C_VEL
LIN {X 0,Y 298.926,Z 358.25,A -85,B 0,C 180,E1 -16471.347,E2 -16471.347} C_VEL
LIN {X 0,Y 298.789,Z 358.264,A -85,B 0,C 180,E1 -16476.754,E2 -16476.754} C_VEL
LIN {X 0,Y 298.681,Z 358.282,A -85,B 0,C 180,E1 -16479.48,E2 -16479.48} C_VEL
LIN {X 0,Y 298.554,Z 358.296,A -85,B 0,C 180,E1 -16483.615,E2 -16483.615} C_VEL
LIN {X 0,Y 298.55,Z 358.293,A -85,B 0,C 180,E1 -16486.408,E2 -16486.408} C_VEL
LIN {X 0,Y 298.512,Z 358.3,A -85,B 0,C 180,E1 -16489.654,E2 -16489.654} C_VEL
LIN {X 0,Y 298.458,Z 358.307,A -85,B 0,C 180,E1 -16493.597,E2 -16493.597} C_VEL
LIN {X 0,Y 298.485,Z 358.302,A -85,B 0,C 180,E1 -16496.574,E2 -16496.574} C_VEL
LIN {X 0,Y 298.416,Z 358.312,A -85,B 0,C 180,E1 -16499.641,E2 -16499.641} C_VEL
LIN {X 0,Y 298.393,Z 358.316,A -85,B 0,C 180,E1 -16502.799,E2 -16502.799} C_VEL
LIN {X 0,Y 298.469,Z 358.308,A -85,B 0,C 180,E1 -16506.813,E2 -16506.813} C_VEL
LIN {X 0,Y 298.499,Z 358.523,A -85,B 0,C 180,E1 -16510.834,E2 -16510.834} C_VEL
LIN {X 0,Y 298.808,Z 359.729,A -85,B 0,C 180,E1 -16511.067,E2 -16511.067} C_VEL
LIN {X 0,Y 302.398,Z 372.043,A -85,B 0,C 180,E1 -16512.374,E2 -16512.374} C_VEL
LIN {X 0,Y 304.797,Z 381.368,A -85,B 0,C 180,E1 -16513.538,E2 -16513.538} C_VEL
LIN {X 0,Y 303.839,Z 392.372,A -85,B 0,C 180,E1 -16514.967,E2 -16514.967} C_VEL
LIN {X 0,Y 302.752,Z 402.368,A -85,B 0,C 180,E1 -16516.551,E2 -16516.551} C_VEL
LIN {X 0,Y 301.831,Z 410.757,A -85,B 0,C 180,E1 -16518.167,E2 -16518.167} C_VEL
LIN {X 0,Y 300.79,Z 419.632,A -85,B 0,C 180,E1 -16520.272,E2 -16520.272} C_VEL
LIN {X 0,Y 299.985,Z 427.057,A -85,B 0,C 180,E1 -16522.474,E2 -16522.474} C_VEL
LIN {X 0,Y 299.343,Z 433.004,A -85,B 0,C 180,E1 -16524.743,E2 -16524.743} C_VEL
LIN {X 0,Y 298.946,Z 437.979,A -85,B 0,C 180,E1 -16527.268,E2 -16527.268} C_VEL
LIN {X 0,Y 298.773,Z 440.242,A -85,B 0,C 180,E1 -16528.835,E2 -16528.835} C_VEL
LIN {X 0,Y 298.743,Z 442.069,A -85,B 0,C 180,E1 -16530.506,E2 -16530.506} C_VEL
LIN {X 0,Y 298.775,Z 443.092,A -85,B 0,C 180,E1 -16531.936,E2 -16531.936} C_VEL
LIN {X 0,Y 298.911,Z 443.726,A -85,B 0,C 180,E1 -16533.466,E2 -16533.466} C_VEL
LIN {X 0,Y 299.186,Z 443.829,A -85,B 0,C 180,E1 -16534.987,E2 -16534.987} C_VEL
LIN {X 0,Y 299.614,Z 443.421,A -85,B 0,C 180,E1 -16536.499,E2 -16536.499} C_VEL
LIN {X 0,Y 300.103,Z 442.554,A -85,B 0,C 180,E1 -16537.994,E2 -16537.994} C_VEL
LIN {X 0,Y 300.708,Z 441.15,A -85,B 0,C 180,E1 -16539.478,E2 -16539.478} C_VEL
